  PROC DrawPart242()
    MoveL Offs(pOrigin,242.99,335.65,0.00),v40,z0,tPen\WObj:=wPaper;
    MoveL Offs(pOrigin,241.50,335.65,0.00),v40,fine,tPen\WObj:=wPaper;
    MoveL Offs(pOrigin,241.50,335.65,6.00),v60,z5,tPen\WObj:=wPaper;
    MoveL Offs(pOrigin,240.78,337.99,6.00),vTravel,z5,tPen\WObj:=wPaper;
    MoveL Offs(pOrigin,240.78,337.99,0.00),v60,z0,tPen\WObj:=wPaper;
    MoveL Offs(pOrigin,240.78,339.05,0.00),v40,z0,tPen\WObj:=wPaper;
    MoveL Offs(pOrigin,239.73,339.05,0.00),v40,z0,tPen\WObj:=wPaper;
    MoveL Offs(pOrigin,239.73,337.99,0.00),v40,fine,tPen\WObj:=wPaper;
    MoveL Offs(pOrigin,239.73,337.99,6.00),v60,z5,tPen\WObj:=wPaper;
    MoveL Offs(pOrigin,237.46,338.14,6.00),vTravel,z5,tPen\WObj:=wPaper;
    MoveL Offs(pOrigin,237.46,338.14,0.00),v60,z0,tPen\WObj:=wPaper;
    MoveL Offs(pOrigin,243.84,338.14,0.00),v40,fine,tPen\WObj:=wPaper;
    MoveL Offs(pOrigin,243.84,338.14,6.00),v60,z5,tPen\WObj:=wPaper;
    MoveL Offs(pOrigin,249.21,337.62,6.00),vTravel,z5,tPen\WObj:=wPaper;
    MoveL Offs(pOrigin,249.21,337.62,0.00),v60,z0,tPen\WObj:=wPaper;
    MoveL Offs(pOrigin,251.17,339.57,0.00),v40,fine,tPen\WObj:=wPaper;
    MoveL Offs(pOrigin,251.17,339.57,6.00),v60,z5,tPen\WObj:=wPaper;
    MoveL Offs(pOrigin,257.20,338.92,6.00),vTravel,z5,tPen\WObj:=wPaper;
    MoveL Offs(pOrigin,257.20,338.92,0.00),v60,z0,tPen\WObj:=wPaper;
    MoveL Offs(pOrigin,264.41,331.71,0.00),v40,fine,tPen\WObj:=wPaper;
    MoveL Offs(pOrigin,264.41,331.71,6.00),v60,z5,tPen\WObj:=wPaper;
    MoveL Offs(pOrigin,262.96,331.61,6.00),vTravel,z5,tPen\WObj:=wPaper;
    MoveL Offs(pOrigin,262.96,331.61,0.00),v60,z0,tPen\WObj:=wPaper;
    MoveL Offs(pOrigin,262.54,331.83,0.00),v40,z0,tPen\WObj:=wPaper;
    MoveL Offs(pOrigin,262.54,332.67,0.00),v40,fine,tPen\WObj:=wPaper;
    MoveL Offs(pOrigin,262.54,332.67,6.00),v60,z5,tPen\WObj:=wPaper;
    MoveL Offs(pOrigin,258.92,334.38,6.00),vTravel,z5,tPen\WObj:=wPaper;
    MoveL Offs(pOrigin,258.92,334.38,0.00),v60,z0,tPen\WObj:=wPaper;
    MoveL Offs(pOrigin,259.14,333.95,0.00),v40,z0,tPen\WObj:=wPaper;
    MoveL Offs(pOrigin,258.92,334.38,0.00),v40,z0,tPen\WObj:=wPaper;
    MoveL Offs(pOrigin,258.49,334.95,0.00),v40,z0,tPen\WObj:=wPaper;
    MoveL Offs(pOrigin,256.69,333.15,0.00),v40,fine,tPen\WObj:=wPaper;
    MoveL Offs(pOrigin,256.69,333.15,6.00),v60,z5,tPen\WObj:=wPaper;
    MoveL Offs(pOrigin,259.60,338.01,6.00),vTravel,z5,tPen\WObj:=wPaper;
    MoveL Offs(pOrigin,259.60,338.01,0.00),v60,z0,tPen\WObj:=wPaper;
    MoveL Offs(pOrigin,274.17,323.44,0.00),v40,fine,tPen\WObj:=wPaper;
    MoveL Offs(pOrigin,274.17,323.44,6.00),v60,z5,tPen\WObj:=wPaper;
    MoveL Offs(pOrigin,279.11,319.08,6.00),vTravel,z5,tPen\WObj:=wPaper;
    MoveL Offs(pOrigin,279.11,319.08,0.00),v60,z0,tPen\WObj:=wPaper;
    MoveL Offs(pOrigin,279.54,319.29,0.00),v40,z0,tPen\WObj:=wPaper;
    MoveL Offs(pOrigin,279.11,319.08,0.00),v40,fine,tPen\WObj:=wPaper;
    MoveL Offs(pOrigin,279.11,319.08,6.00),v60,z5,tPen\WObj:=wPaper;
    MoveL Offs(pOrigin,282.73,312.27,6.00),vTravel,z5,tPen\WObj:=wPaper;
    MoveL Offs(pOrigin,282.73,312.27,0.00),v60,z0,tPen\WObj:=wPaper;
    MoveL Offs(pOrigin,285.70,312.06,0.00),v40,z0,tPen\WObj:=wPaper;
    MoveL Offs(pOrigin,285.98,311.67,0.00),v40,z0,tPen\WObj:=wPaper;
    MoveL Offs(pOrigin,287.19,312.87,0.00),v40,z0,tPen\WObj:=wPaper;
    MoveL Offs(pOrigin,286.29,313.46,0.00),v40,z0,tPen\WObj:=wPaper;
    MoveL Offs(pOrigin,285.54,312.71,0.00),v40,fine,tPen\WObj:=wPaper;
    MoveL Offs(pOrigin,285.54,312.71,6.00),v60,z5,tPen\WObj:=wPaper;
    MoveL Offs(pOrigin,287.03,309.72,6.00),vTravel,z5,tPen\WObj:=wPaper;
    MoveL Offs(pOrigin,287.03,309.72,0.00),v60,z0,tPen\WObj:=wPaper;
    MoveL Offs(pOrigin,291.83,314.53,0.00),v40,fine,tPen\WObj:=wPaper;
    MoveL Offs(pOrigin,291.83,314.53,6.00),v60,z5,tPen\WObj:=wPaper;
    MoveL Offs(pOrigin,291.86,312.79,6.00),vTravel,z5,tPen\WObj:=wPaper;
    MoveL Offs(pOrigin,291.86,312.79,0.00),v60,z0,tPen\WObj:=wPaper;
    MoveL Offs(pOrigin,289.52,312.79,0.00),v40,z0,tPen\WObj:=wPaper;
    MoveL Offs(pOrigin,289.52,312.06,0.00),v40,z0,tPen\WObj:=wPaper;
    MoveL Offs(pOrigin,289.31,312.49,0.00),v40,z0,tPen\WObj:=wPaper;
    MoveL Offs(pOrigin,289.52,312.06,0.00),v40,z0,tPen\WObj:=wPaper;
    MoveL Offs(pOrigin,288.67,311.42,0.00),v40,z0,tPen\WObj:=wPaper;
    MoveL Offs(pOrigin,288.46,311.85,0.00),v40,z0,tPen\WObj:=wPaper;
    MoveL Offs(pOrigin,288.67,311.42,0.00),v40,fine,tPen\WObj:=wPaper;
    MoveL Offs(pOrigin,288.67,311.42,6.00),v60,z5,tPen\WObj:=wPaper;
    MoveL Offs(pOrigin,280.81,308.45,6.00),vTravel,z5,tPen\WObj:=wPaper;
    MoveL Offs(pOrigin,280.81,308.45,0.00),v60,z0,tPen\WObj:=wPaper;
    MoveL Offs(pOrigin,280.17,308.66,0.00),v40,z0,tPen\WObj:=wPaper;
    MoveL Offs(pOrigin,279.75,309.30,0.00),v40,z0,tPen\WObj:=wPaper;
    MoveL Offs(pOrigin,279.75,309.30,0.00),v40,z0,tPen\WObj:=wPaper;
    MoveL Offs(pOrigin,278.48,308.88,0.00),v40,z0,tPen\WObj:=wPaper;
    MoveL Offs(pOrigin,278.69,307.60,0.00),v40,z0,tPen\WObj:=wPaper;
    MoveL Offs(pOrigin,279.54,307.51,0.00),v40,z0,tPen\WObj:=wPaper;
    MoveL Offs(pOrigin,270.61,307.51,0.00),v40,fine,tPen\WObj:=wPaper;
    MoveL Offs(pOrigin,270.61,307.51,6.00),v60,z5,tPen\WObj:=wPaper;
    MoveL Offs(pOrigin,273.80,305.40,6.00),vTravel,z5,tPen\WObj:=wPaper;
    MoveL Offs(pOrigin,273.80,305.40,0.00),v60,z0,tPen\WObj:=wPaper;
    MoveL Offs(pOrigin,279.54,305.40,0.00),v40,z0,tPen\WObj:=wPaper;
    MoveL Offs(pOrigin,279.75,304.34,0.00),v40,z0,tPen\WObj:=wPaper;
    MoveL Offs(pOrigin,274.23,304.34,0.00),v40,fine,tPen\WObj:=wPaper;
    MoveL Offs(pOrigin,274.23,304.34,6.00),v60,z5,tPen\WObj:=wPaper;
    MoveL Offs(pOrigin,274.27,302.94,6.00),vTravel,z5,tPen\WObj:=wPaper;
    MoveL Offs(pOrigin,274.27,302.94,0.00),v60,z0,tPen\WObj:=wPaper;
    MoveL Offs(pOrigin,280.28,308.95,0.00),v40,fine,tPen\WObj:=wPaper;
    MoveL Offs(pOrigin,280.28,308.95,6.00),v60,z5,tPen\WObj:=wPaper;
    MoveL Offs(pOrigin,278.80,303.35,6.00),vTravel,z5,tPen\WObj:=wPaper;
    MoveL Offs(pOrigin,278.80,303.35,0.00),v60,z0,tPen\WObj:=wPaper;
    MoveL Offs(pOrigin,278.80,301.86,0.00),v40,fine,tPen\WObj:=wPaper;
    MoveL Offs(pOrigin,278.80,301.86,6.00),v60,z5,tPen\WObj:=wPaper;
    MoveL Offs(pOrigin,276.77,302.71,6.00),vTravel,z5,tPen\WObj:=wPaper;
    MoveL Offs(pOrigin,276.77,302.71,0.00),v60,z0,tPen\WObj:=wPaper;
    MoveL Offs(pOrigin,276.56,304.41,0.00),v40,fine,tPen\WObj:=wPaper;
    MoveL Offs(pOrigin,276.56,304.41,6.00),v60,z5,tPen\WObj:=wPaper;
    MoveL Offs(pOrigin,264.66,324.60,6.00),vTravel,z5,tPen\WObj:=wPaper;
    MoveL Offs(pOrigin,264.66,324.60,0.00),v60,z0,tPen\WObj:=wPaper;
    MoveL Offs(pOrigin,265.09,325.24,0.00),v40,z0,tPen\WObj:=wPaper;
    MoveL Offs(pOrigin,264.66,324.60,0.00),v40,fine,tPen\WObj:=wPaper;
    MoveL Offs(pOrigin,264.66,324.60,6.00),v60,z5,tPen\WObj:=wPaper;
    MoveL Offs(pOrigin,247.24,328.17,6.00),vTravel,z5,tPen\WObj:=wPaper;
    MoveL Offs(pOrigin,247.24,328.17,0.00),v60,z0,tPen\WObj:=wPaper;
    MoveL Offs(pOrigin,232.66,313.60,0.00),v40,fine,tPen\WObj:=wPaper;
    MoveL Offs(pOrigin,232.66,313.60,6.00),v60,z5,tPen\WObj:=wPaper;
    MoveL Offs(pOrigin,231.09,314.90,6.00),vTravel,z5,tPen\WObj:=wPaper;
    MoveL Offs(pOrigin,231.09,314.90,0.00),v60,z0,tPen\WObj:=wPaper;
    MoveL Offs(pOrigin,216.64,314.90,0.00),v40,z0,tPen\WObj:=wPaper;
    MoveL Offs(pOrigin,216.64,315.67,0.00),v40,z0,tPen\WObj:=wPaper;
    MoveL Offs(pOrigin,216.00,316.10,0.00),v40,z0,tPen\WObj:=wPaper;
    MoveL Offs(pOrigin,215.72,317.38,0.00),v40,z0,tPen\WObj:=wPaper;
    MoveL Offs(pOrigin,215.15,317.80,0.00),v40,fine,tPen\WObj:=wPaper;
    MoveL Offs(pOrigin,215.15,317.80,6.00),v60,z5,tPen\WObj:=wPaper;
    MoveL Offs(pOrigin,213.95,317.29,6.00),vTravel,z5,tPen\WObj:=wPaper;
    MoveL Offs(pOrigin,213.95,317.29,0.00),v60,z0,tPen\WObj:=wPaper;
    MoveL Offs(pOrigin,210.34,313.68,0.00),v40,z0,tPen\WObj:=wPaper;
    MoveL Offs(pOrigin,210.05,313.76,0.00),v40,z0,tPen\WObj:=wPaper;
    MoveL Offs(pOrigin,209.62,314.19,0.00),v40,z0,tPen\WObj:=wPaper;
    MoveL Offs(pOrigin,210.05,313.76,0.00),v40,fine,tPen\WObj:=wPaper;
    MoveL Offs(pOrigin,210.05,313.76,6.00),v60,z5,tPen\WObj:=wPaper;
    MoveL Offs(pOrigin,210.90,312.91,6.00),vTravel,z5,tPen\WObj:=wPaper;
    MoveL Offs(pOrigin,210.90,312.91,0.00),v60,z0,tPen\WObj:=wPaper;
    MoveL Offs(pOrigin,210.26,313.55,0.00),v40,z0,tPen\WObj:=wPaper;
    MoveL Offs(pOrigin,210.90,312.91,0.00),v40,z0,tPen\WObj:=wPaper;
  ENDPROC

  PROC DrawPart243()
    MoveL Offs(pOrigin,210.94,312.78,0.00),v40,z0,tPen\WObj:=wPaper;
    MoveL Offs(pOrigin,214.69,316.54,0.00),v40,fine,tPen\WObj:=wPaper;
    MoveL Offs(pOrigin,214.69,316.54,6.00),v60,z5,tPen\WObj:=wPaper;
    MoveL Offs(pOrigin,213.45,317.02,6.00),vTravel,z5,tPen\WObj:=wPaper;
    MoveL Offs(pOrigin,213.45,317.02,0.00),v60,z0,tPen\WObj:=wPaper;
    MoveL Offs(pOrigin,212.39,317.02,0.00),v40,z0,tPen\WObj:=wPaper;
    MoveL Offs(pOrigin,211.85,316.68,0.00),v40,z0,tPen\WObj:=wPaper;
    MoveL Offs(pOrigin,213.50,318.33,0.00),v40,z0,tPen\WObj:=wPaper;
    MoveL Offs(pOrigin,213.24,318.07,0.00),v40,z0,tPen\WObj:=wPaper;
    MoveL Offs(pOrigin,211.96,318.07,0.00),v40,z0,tPen\WObj:=wPaper;
    MoveL Offs(pOrigin,211.55,317.88,0.00),v40,z0,tPen\WObj:=wPaper;
    MoveL Offs(pOrigin,213.21,319.53,0.00),v40,z0,tPen\WObj:=wPaper;
    MoveL Offs(pOrigin,212.81,319.13,0.00),v40,z0,tPen\WObj:=wPaper;
    MoveL Offs(pOrigin,211.32,319.13,0.00),v40,z0,tPen\WObj:=wPaper;
    MoveL Offs(pOrigin,211.32,319.08,0.00),v40,z0,tPen\WObj:=wPaper;
    MoveL Offs(pOrigin,211.54,318.65,0.00),v40,z0,tPen\WObj:=wPaper;
    MoveL Offs(pOrigin,211.32,319.08,0.00),v40,z0,tPen\WObj:=wPaper;
    MoveL Offs(pOrigin,210.96,318.77,0.00),v40,z0,tPen\WObj:=wPaper;
    MoveL Offs(pOrigin,212.76,320.58,0.00),v40,fine,tPen\WObj:=wPaper;
    MoveL Offs(pOrigin,212.76,320.58,6.00),v60,z5,tPen\WObj:=wPaper;
    MoveL Offs(pOrigin,210.21,323.19,6.00),vTravel,z5,tPen\WObj:=wPaper;
    MoveL Offs(pOrigin,210.21,323.19,0.00),v60,z0,tPen\WObj:=wPaper;
    MoveL Offs(pOrigin,204.35,329.05,0.00),v40,fine,tPen\WObj:=wPaper;
    MoveL Offs(pOrigin,204.35,329.05,6.00),v60,z5,tPen\WObj:=wPaper;
    MoveL Offs(pOrigin,208.05,327.15,6.00),vTravel,z5,tPen\WObj:=wPaper;
    MoveL Offs(pOrigin,208.05,327.15,0.00),v60,z0,tPen\WObj:=wPaper;
    MoveL Offs(pOrigin,208.05,325.88,0.00),v40,fine,tPen\WObj:=wPaper;
    MoveL Offs(pOrigin,208.05,325.88,6.00),v60,z5,tPen\WObj:=wPaper;
    MoveL Offs(pOrigin,209.10,326.51,6.00),vTravel,z5,tPen\WObj:=wPaper;
    MoveL Offs(pOrigin,209.10,326.51,0.00),v60,z0,tPen\WObj:=wPaper;
    MoveL Offs(pOrigin,209.10,327.58,0.00),v40,fine,tPen\WObj:=wPaper;
    MoveL Offs(pOrigin,209.10,327.58,6.00),v60,z5,tPen\WObj:=wPaper;
    MoveL Offs(pOrigin,210.26,329.06,6.00),vTravel,z5,tPen\WObj:=wPaper;
    MoveL Offs(pOrigin,210.26,329.06,0.00),v60,z0,tPen\WObj:=wPaper;
    MoveL Offs(pOrigin,210.69,329.49,0.00),v40,z0,tPen\WObj:=wPaper;
    MoveL Offs(pOrigin,210.26,329.06,0.00),v40,fine,tPen\WObj:=wPaper;
    MoveL Offs(pOrigin,210.26,329.06,6.00),v60,z5,tPen\WObj:=wPaper;
    MoveL Offs(pOrigin,209.41,325.66,6.00),vTravel,z5,tPen\WObj:=wPaper;
    MoveL Offs(pOrigin,209.41,325.66,0.00),v60,z0,tPen\WObj:=wPaper;
    MoveL Offs(pOrigin,209.84,326.09,0.00),v40,z0,tPen\WObj:=wPaper;
    MoveL Offs(pOrigin,209.41,325.66,0.00),v40,z0,tPen\WObj:=wPaper;
    MoveL Offs(pOrigin,209.93,325.21,0.00),v40,z0,tPen\WObj:=wPaper;
    MoveL Offs(pOrigin,209.03,324.31,0.00),v40,fine,tPen\WObj:=wPaper;
    MoveL Offs(pOrigin,209.03,324.31,6.00),v60,z5,tPen\WObj:=wPaper;
    MoveL Offs(pOrigin,214.88,327.18,6.00),vTravel,z5,tPen\WObj:=wPaper;
    MoveL Offs(pOrigin,214.88,327.18,0.00),v60,z0,tPen\WObj:=wPaper;
    MoveL Offs(pOrigin,217.13,329.43,0.00),v40,fine,tPen\WObj:=wPaper;
    MoveL Offs(pOrigin,217.13,329.43,6.00),v60,z5,tPen\WObj:=wPaper;
    MoveL Offs(pOrigin,219.38,328.69,6.00),vTravel,z5,tPen\WObj:=wPaper;
    MoveL Offs(pOrigin,219.38,328.69,0.00),v60,z0,tPen\WObj:=wPaper;
    MoveL Offs(pOrigin,217.72,327.03,0.00),v40,fine,tPen\WObj:=wPaper;
    MoveL Offs(pOrigin,217.72,327.03,6.00),v60,z5,tPen\WObj:=wPaper;
    MoveL Offs(pOrigin,220.68,328.42,6.00),vTravel,z5,tPen\WObj:=wPaper;
    MoveL Offs(pOrigin,220.68,328.42,0.00),v60,z0,tPen\WObj:=wPaper;
    MoveL Offs(pOrigin,221.10,328.21,0.00),v40,z0,tPen\WObj:=wPaper;
    MoveL Offs(pOrigin,220.68,328.42,0.00),v40,fine,tPen\WObj:=wPaper;
    MoveL Offs(pOrigin,220.68,328.42,6.00),v60,z5,tPen\WObj:=wPaper;
    MoveL Offs(pOrigin,223.12,329.45,6.00),vTravel,z5,tPen\WObj:=wPaper;
    MoveL Offs(pOrigin,223.12,329.45,0.00),v60,z0,tPen\WObj:=wPaper;
    MoveL Offs(pOrigin,224.17,330.50,0.00),v40,z0,tPen\WObj:=wPaper;
    MoveL Offs(pOrigin,224.77,329.60,0.00),v40,z0,tPen\WObj:=wPaper;
    MoveL Offs(pOrigin,223.87,328.70,0.00),v40,z0,tPen\WObj:=wPaper;
    MoveL Offs(pOrigin,224.71,329.06,0.00),v40,z0,tPen\WObj:=wPaper;
    MoveL Offs(pOrigin,223.44,329.06,0.00),v40,z0,tPen\WObj:=wPaper;
    MoveL Offs(pOrigin,219.61,330.55,0.00),v40,z0,tPen\WObj:=wPaper;
    MoveL Offs(pOrigin,216.21,330.76,0.00),v40,z0,tPen\WObj:=wPaper;
    MoveL Offs(pOrigin,215.86,330.98,0.00),v40,z0,tPen\WObj:=wPaper;
    MoveL Offs(pOrigin,215.79,331.61,0.00),v40,fine,tPen\WObj:=wPaper;
    MoveL Offs(pOrigin,215.79,331.61,6.00),v60,z5,tPen\WObj:=wPaper;
    MoveL Offs(pOrigin,215.58,332.86,6.00),vTravel,z5,tPen\WObj:=wPaper;
    MoveL Offs(pOrigin,215.58,332.86,0.00),v60,z0,tPen\WObj:=wPaper;
    MoveL Offs(pOrigin,214.51,332.86,0.00),v40,fine,tPen\WObj:=wPaper;
    MoveL Offs(pOrigin,214.51,332.86,6.00),v60,z5,tPen\WObj:=wPaper;
    MoveL Offs(pOrigin,209.20,333.52,6.00),vTravel,z5,tPen\WObj:=wPaper;
    MoveL Offs(pOrigin,209.20,333.52,0.00),v60,z0,tPen\WObj:=wPaper;
    MoveL Offs(pOrigin,209.62,333.74,0.00),v40,z0,tPen\WObj:=wPaper;
    MoveL Offs(pOrigin,209.20,333.52,0.00),v40,fine,tPen\WObj:=wPaper;
    MoveL Offs(pOrigin,209.20,333.52,6.00),v60,z5,tPen\WObj:=wPaper;
    MoveL Offs(pOrigin,218.86,336.94,6.00),vTravel,z5,tPen\WObj:=wPaper;
    MoveL Offs(pOrigin,218.86,336.94,0.00),v60,z0,tPen\WObj:=wPaper;
    MoveL Offs(pOrigin,226.67,329.13,0.00),v40,z0,tPen\WObj:=wPaper;
    MoveL Offs(pOrigin,227.05,328.00,0.00),v40,z0,tPen\WObj:=wPaper;
    MoveL Offs(pOrigin,227.26,327.58,0.00),v40,z0,tPen\WObj:=wPaper;
    MoveL Offs(pOrigin,227.05,328.00,0.00),v40,fine,tPen\WObj:=wPaper;
    MoveL Offs(pOrigin,227.05,328.00,6.00),v60,z5,tPen\WObj:=wPaper;
    MoveL Offs(pOrigin,228.02,329.27,6.00),vTravel,z5,tPen\WObj:=wPaper;
    MoveL Offs(pOrigin,228.02,329.27,0.00),v60,z0,tPen\WObj:=wPaper;
    MoveL Offs(pOrigin,220.20,337.09,0.00),v40,fine,tPen\WObj:=wPaper;
    MoveL Offs(pOrigin,220.20,337.09,6.00),v60,z5,tPen\WObj:=wPaper;
    MoveL Offs(pOrigin,226.41,336.02,6.00),vTravel,z5,tPen\WObj:=wPaper;
    MoveL Offs(pOrigin,226.41,336.02,0.00),v60,z0,tPen\WObj:=wPaper;
    MoveL Offs(pOrigin,232.79,336.02,0.00),v40,fine,tPen\WObj:=wPaper;
    MoveL Offs(pOrigin,232.79,336.02,6.00),v60,z5,tPen\WObj:=wPaper;
    MoveL Offs(pOrigin,233.10,333.15,6.00),vTravel,z5,tPen\WObj:=wPaper;
    MoveL Offs(pOrigin,233.10,333.15,0.00),v60,z0,tPen\WObj:=wPaper;
    MoveL Offs(pOrigin,226.64,339.61,0.00),v40,fine,tPen\WObj:=wPaper;
    MoveL Offs(pOrigin,226.64,339.61,6.00),v60,z5,tPen\WObj:=wPaper;
    MoveL Offs(pOrigin,226.00,333.31,6.00),vTravel,z5,tPen\WObj:=wPaper;
    MoveL Offs(pOrigin,226.00,333.31,0.00),v60,z0,tPen\WObj:=wPaper;
    MoveL Offs(pOrigin,226.00,332.04,0.00),v40,z0,tPen\WObj:=wPaper;
    MoveL Offs(pOrigin,226.27,331.11,0.00),v40,z0,tPen\WObj:=wPaper;
    MoveL Offs(pOrigin,228.38,333.21,0.00),v40,fine,tPen\WObj:=wPaper;
    MoveL Offs(pOrigin,228.38,333.21,6.00),v60,z5,tPen\WObj:=wPaper;
    MoveL Offs(pOrigin,224.73,326.59,6.00),vTravel,z5,tPen\WObj:=wPaper;
    MoveL Offs(pOrigin,224.73,326.59,0.00),v60,z0,tPen\WObj:=wPaper;
    MoveL Offs(pOrigin,240.51,310.81,0.00),v40,fine,tPen\WObj:=wPaper;
    MoveL Offs(pOrigin,240.51,310.81,6.00),v60,z5,tPen\WObj:=wPaper;
    MoveL Offs(pOrigin,238.20,313.17,6.00),vTravel,z5,tPen\WObj:=wPaper;
    MoveL Offs(pOrigin,238.20,313.17,0.00),v60,z0,tPen\WObj:=wPaper;
    MoveL Offs(pOrigin,239.25,314.22,0.00),v40,fine,tPen\WObj:=wPaper;
    MoveL Offs(pOrigin,239.25,314.22,6.00),v60,z5,tPen\WObj:=wPaper;
    MoveL Offs(pOrigin,244.19,313.18,6.00),vTravel,z5,tPen\WObj:=wPaper;
    MoveL Offs(pOrigin,244.19,313.18,0.00),v60,z0,tPen\WObj:=wPaper;
    MoveL Offs(pOrigin,245.25,314.24,0.00),v40,fine,tPen\WObj:=wPaper;
    MoveL Offs(pOrigin,245.25,314.24,6.00),v60,z5,tPen\WObj:=wPaper;
    MoveL Offs(pOrigin,234.45,320.77,6.00),vTravel,z5,tPen\WObj:=wPaper;
    MoveL Offs(pOrigin,234.45,320.77,0.00),v60,z0,tPen\WObj:=wPaper;
    MoveL Offs(pOrigin,234.45,322.90,0.00),v40,fine,tPen\WObj:=wPaper;
    MoveL Offs(pOrigin,234.45,322.90,6.00),v60,z5,tPen\WObj:=wPaper;
    MoveL Offs(pOrigin,233.00,318.07,6.00),vTravel,z5,tPen\WObj:=wPaper;
  ENDPROC

  PROC DrawPart244()
    MoveL Offs(pOrigin,233.00,318.07,0.00),v60,z0,tPen\WObj:=wPaper;
    MoveL Offs(pOrigin,217.91,318.07,0.00),v40,z0,tPen\WObj:=wPaper;
    MoveL Offs(pOrigin,217.70,317.02,0.00),v40,z0,tPen\WObj:=wPaper;
    MoveL Offs(pOrigin,231.94,317.02,0.00),v40,z0,tPen\WObj:=wPaper;
    MoveL Offs(pOrigin,231.30,317.80,0.00),v40,z0,tPen\WObj:=wPaper;
    MoveL Offs(pOrigin,231.09,316.52,0.00),v40,z0,tPen\WObj:=wPaper;
    MoveL Offs(pOrigin,230.45,316.10,0.00),v40,fine,tPen\WObj:=wPaper;
    MoveL Offs(pOrigin,230.45,316.10,6.00),v60,z5,tPen\WObj:=wPaper;
    MoveL Offs(pOrigin,226.00,314.82,6.00),vTravel,z5,tPen\WObj:=wPaper;
    MoveL Offs(pOrigin,226.00,314.82,0.00),v60,z0,tPen\WObj:=wPaper;
    MoveL Offs(pOrigin,226.00,317.80,0.00),v40,fine,tPen\WObj:=wPaper;
    MoveL Offs(pOrigin,226.00,317.80,6.00),v60,z5,tPen\WObj:=wPaper;
    MoveL Offs(pOrigin,221.31,313.34,6.00),vTravel,z5,tPen\WObj:=wPaper;
    MoveL Offs(pOrigin,221.31,313.34,0.00),v60,z0,tPen\WObj:=wPaper;
    MoveL Offs(pOrigin,221.74,312.06,0.00),v40,z0,tPen\WObj:=wPaper;
    MoveL Offs(pOrigin,221.52,311.71,0.00),v40,z0,tPen\WObj:=wPaper;
    MoveL Offs(pOrigin,220.46,312.06,0.00),v40,z0,tPen\WObj:=wPaper;
    MoveL Offs(pOrigin,219.61,313.34,0.00),v40,fine,tPen\WObj:=wPaper;
    MoveL Offs(pOrigin,219.61,313.34,6.00),v60,z5,tPen\WObj:=wPaper;
    MoveL Offs(pOrigin,216.64,313.98,6.00),vTravel,z5,tPen\WObj:=wPaper;
    MoveL Offs(pOrigin,216.64,313.98,0.00),v60,z0,tPen\WObj:=wPaper;
    MoveL Offs(pOrigin,215.57,313.55,0.00),v40,z0,tPen\WObj:=wPaper;
    MoveL Offs(pOrigin,215.57,313.55,0.00),v40,z0,tPen\WObj:=wPaper;
    MoveL Offs(pOrigin,216.00,312.06,0.00),v40,z0,tPen\WObj:=wPaper;
    MoveL Offs(pOrigin,216.64,311.64,0.00),v40,z0,tPen\WObj:=wPaper;
    MoveL Offs(pOrigin,216.21,312.06,0.00),v40,z0,tPen\WObj:=wPaper;
    MoveL Offs(pOrigin,216.64,311.64,0.00),v40,z0,tPen\WObj:=wPaper;
    MoveL Offs(pOrigin,216.21,312.06,0.00),v40,z0,tPen\WObj:=wPaper;
    MoveL Offs(pOrigin,215.44,311.64,0.00),v40,z0,tPen\WObj:=wPaper;
    MoveL Offs(pOrigin,215.44,309.30,0.00),v40,z0,tPen\WObj:=wPaper;
    MoveL Offs(pOrigin,216.49,308.88,0.00),v40,z0,tPen\WObj:=wPaper;
    MoveL Offs(pOrigin,216.49,311.00,0.00),v40,fine,tPen\WObj:=wPaper;
    MoveL Offs(pOrigin,216.49,311.00,6.00),v60,z5,tPen\WObj:=wPaper;
    MoveL Offs(pOrigin,214.38,310.79,6.00),vTravel,z5,tPen\WObj:=wPaper;
    MoveL Offs(pOrigin,214.38,310.79,0.00),v60,z0,tPen\WObj:=wPaper;
    MoveL Offs(pOrigin,214.38,313.12,0.00),v40,fine,tPen\WObj:=wPaper;
    MoveL Offs(pOrigin,214.38,313.12,6.00),v60,z5,tPen\WObj:=wPaper;
    MoveL Offs(pOrigin,213.33,309.30,6.00),vTravel,z5,tPen\WObj:=wPaper;
    MoveL Offs(pOrigin,213.33,309.30,0.00),v60,z0,tPen\WObj:=wPaper;
    MoveL Offs(pOrigin,213.33,306.96,0.00),v40,z0,tPen\WObj:=wPaper;
    MoveL Offs(pOrigin,212.27,306.75,0.00),v40,z0,tPen\WObj:=wPaper;
    MoveL Offs(pOrigin,212.27,308.66,0.00),v40,z0,tPen\WObj:=wPaper;
    MoveL Offs(pOrigin,211.21,308.45,0.00),v40,z0,tPen\WObj:=wPaper;
    MoveL Offs(pOrigin,211.21,306.32,0.00),v40,z0,tPen\WObj:=wPaper;
    MoveL Offs(pOrigin,210.69,306.96,0.00),v40,z0,tPen\WObj:=wPaper;
    MoveL Offs(pOrigin,211.96,306.75,0.00),v40,z0,tPen\WObj:=wPaper;
    MoveL Offs(pOrigin,212.81,305.97,0.00),v40,z0,tPen\WObj:=wPaper;
    MoveL Offs(pOrigin,213.88,305.69,0.00),v40,fine,tPen\WObj:=wPaper;
    MoveL Offs(pOrigin,213.88,305.69,6.00),v60,z5,tPen\WObj:=wPaper;
    MoveL Offs(pOrigin,211.96,303.35,6.00),vTravel,z5,tPen\WObj:=wPaper;
    MoveL Offs(pOrigin,211.96,303.35,0.00),v60,z0,tPen\WObj:=wPaper;
    MoveL Offs(pOrigin,211.47,301.86,0.00),v40,z0,tPen\WObj:=wPaper;
    MoveL Offs(pOrigin,209.84,301.01,0.00),v40,z0,tPen\WObj:=wPaper;
    MoveL Offs(pOrigin,209.84,301.01,0.00),v40,z0,tPen\WObj:=wPaper;
    MoveL Offs(pOrigin,207.93,300.66,0.00),v40,z0,tPen\WObj:=wPaper;
    MoveL Offs(pOrigin,207.29,300.02,0.00),v40,z0,tPen\WObj:=wPaper;
    MoveL Offs(pOrigin,205.80,300.23,0.00),v40,z0,tPen\WObj:=wPaper;
    MoveL Offs(pOrigin,202.82,298.53,0.00),v40,z0,tPen\WObj:=wPaper;
    MoveL Offs(pOrigin,202.40,298.89,0.00),v40,z0,tPen\WObj:=wPaper;
    MoveL Offs(pOrigin,202.40,299.95,0.00),v40,z0,tPen\WObj:=wPaper;
    MoveL Offs(pOrigin,203.04,300.12,0.00),v40,z0,tPen\WObj:=wPaper;
    MoveL Offs(pOrigin,208.78,300.12,0.00),v40,fine,tPen\WObj:=wPaper;
    MoveL Offs(pOrigin,208.78,300.12,6.00),v60,z5,tPen\WObj:=wPaper;
    MoveL Offs(pOrigin,209.84,301.01,6.00),vTravel,z5,tPen\WObj:=wPaper;
    MoveL Offs(pOrigin,209.84,301.01,0.00),v60,z0,tPen\WObj:=wPaper;
    MoveL Offs(pOrigin,209.34,298.89,0.00),v40,z0,tPen\WObj:=wPaper;
    MoveL Offs(pOrigin,207.50,296.76,0.00),v40,fine,tPen\WObj:=wPaper;
    MoveL Offs(pOrigin,207.50,296.76,6.00),v60,z5,tPen\WObj:=wPaper;
    MoveL Offs(pOrigin,205.59,302.92,6.00),vTravel,z5,tPen\WObj:=wPaper;
    MoveL Offs(pOrigin,205.59,302.92,0.00),v60,z0,tPen\WObj:=wPaper;
    MoveL Offs(pOrigin,206.65,303.14,0.00),v40,z0,tPen\WObj:=wPaper;
    MoveL Offs(pOrigin,206.86,303.77,0.00),v40,fine,tPen\WObj:=wPaper;
    MoveL Offs(pOrigin,206.86,303.77,6.00),v60,z5,tPen\WObj:=wPaper;
    MoveL Offs(pOrigin,202.24,308.56,6.00),vTravel,z5,tPen\WObj:=wPaper;
    MoveL Offs(pOrigin,202.24,308.56,0.00),v60,z0,tPen\WObj:=wPaper;
    MoveL Offs(pOrigin,200.13,306.46,0.00),v40,z0,tPen\WObj:=wPaper;
    MoveL Offs(pOrigin,199.21,306.46,0.00),v40,z0,tPen\WObj:=wPaper;
    MoveL Offs(pOrigin,197.51,306.46,0.00),v40,fine,tPen\WObj:=wPaper;
    MoveL Offs(pOrigin,197.51,306.46,6.00),v60,z5,tPen\WObj:=wPaper;
    MoveL Offs(pOrigin,199.64,300.59,6.00),vTravel,z5,tPen\WObj:=wPaper;
    MoveL Offs(pOrigin,199.64,300.59,0.00),v60,z0,tPen\WObj:=wPaper;
    MoveL Offs(pOrigin,200.06,300.80,0.00),v40,z0,tPen\WObj:=wPaper;
    MoveL Offs(pOrigin,199.64,300.59,0.00),v40,fine,tPen\WObj:=wPaper;
    MoveL Offs(pOrigin,199.64,300.59,6.00),v60,z5,tPen\WObj:=wPaper;
    MoveL Offs(pOrigin,207.95,315.77,6.00),vTravel,z5,tPen\WObj:=wPaper;
    MoveL Offs(pOrigin,207.95,315.77,0.00),v60,z0,tPen\WObj:=wPaper;
    MoveL Offs(pOrigin,209.00,316.82,0.00),v40,z0,tPen\WObj:=wPaper;
    MoveL Offs(pOrigin,209.20,316.95,0.00),v40,z0,tPen\WObj:=wPaper;
    MoveL Offs(pOrigin,208.92,317.52,0.00),v40,z0,tPen\WObj:=wPaper;
    MoveL Offs(pOrigin,207.50,318.01,0.00),v40,z0,tPen\WObj:=wPaper;
    MoveL Offs(pOrigin,205.59,318.23,0.00),v40,z0,tPen\WObj:=wPaper;
    MoveL Offs(pOrigin,202.19,317.80,0.00),v40,z0,tPen\WObj:=wPaper;
    MoveL Offs(pOrigin,201.76,318.01,0.00),v40,fine,tPen\WObj:=wPaper;
    MoveL Offs(pOrigin,201.76,318.01,6.00),v60,z5,tPen\WObj:=wPaper;
    MoveL Offs(pOrigin,219.66,319.29,6.00),vTravel,z5,tPen\WObj:=wPaper;
    MoveL Offs(pOrigin,219.66,319.29,0.00),v60,z0,tPen\WObj:=wPaper;
    MoveL Offs(pOrigin,219.66,309.94,0.00),v40,fine,tPen\WObj:=wPaper;
    MoveL Offs(pOrigin,219.66,309.94,6.00),v60,z5,tPen\WObj:=wPaper;
    MoveL Offs(pOrigin,222.65,271.92,6.00),vTravel,z5,tPen\WObj:=wPaper;
    MoveL Offs(pOrigin,222.65,271.92,0.00),v60,z0,tPen\WObj:=wPaper;
    MoveL Offs(pOrigin,238.28,256.29,0.00),v40,fine,tPen\WObj:=wPaper;
    MoveL Offs(pOrigin,238.28,256.29,6.00),v60,z5,tPen\WObj:=wPaper;
    MoveL Offs(pOrigin,237.09,254.50,6.00),vTravel,z5,tPen\WObj:=wPaper;
    MoveL Offs(pOrigin,237.09,254.50,0.00),v60,z0,tPen\WObj:=wPaper;
    MoveL Offs(pOrigin,234.68,256.90,0.00),v40,z0,tPen\WObj:=wPaper;
    MoveL Offs(pOrigin,233.93,257.65,0.00),v40,z0,tPen\WObj:=wPaper;
    MoveL Offs(pOrigin,220.26,271.32,0.00),v40,z0,tPen\WObj:=wPaper;
    MoveL Offs(pOrigin,219.95,271.02,0.00),v40,z0,tPen\WObj:=wPaper;
    MoveL Offs(pOrigin,212.74,263.80,0.00),v40,z0,tPen\WObj:=wPaper;
    MoveL Offs(pOrigin,212.19,264.46,0.00),v40,z0,tPen\WObj:=wPaper;
    MoveL Offs(pOrigin,213.99,262.66,0.00),v40,z0,tPen\WObj:=wPaper;
    MoveL Offs(pOrigin,213.39,261.76,0.00),v40,z0,tPen\WObj:=wPaper;
    MoveL Offs(pOrigin,212.04,263.11,0.00),v40,fine,tPen\WObj:=wPaper;
    MoveL Offs(pOrigin,212.04,263.11,6.00),v60,z5,tPen\WObj:=wPaper;
    MoveL Offs(pOrigin,214.00,259.66,6.00),vTravel,z5,tPen\WObj:=wPaper;
    MoveL Offs(pOrigin,214.00,259.66,0.00),v60,z0,tPen\WObj:=wPaper;
    MoveL Offs(pOrigin,215.95,257.71,0.00),v40,fine,tPen\WObj:=wPaper;
    MoveL Offs(pOrigin,215.95,257.71,6.00),v60,z5,tPen\WObj:=wPaper;
    MoveL Offs(pOrigin,215.36,259.15,6.00),vTravel,z5,tPen\WObj:=wPaper;
    MoveL Offs(pOrigin,215.36,259.15,0.00),v60,z0,tPen\WObj:=wPaper;
  ENDPROC

  PROC DrawPart245()
    MoveL Offs(pOrigin,216.21,259.58,0.00),v40,z0,tPen\WObj:=wPaper;
    MoveL Offs(pOrigin,216.85,259.99,0.00),v40,z0,tPen\WObj:=wPaper;
    MoveL Offs(pOrigin,218.34,259.99,0.00),v40,z0,tPen\WObj:=wPaper;
    MoveL Offs(pOrigin,217.91,259.58,0.00),v40,z0,tPen\WObj:=wPaper;
    MoveL Offs(pOrigin,218.34,260.00,0.00),v40,z0,tPen\WObj:=wPaper;
    MoveL Offs(pOrigin,217.91,259.58,0.00),v40,fine,tPen\WObj:=wPaper;
    MoveL Offs(pOrigin,217.91,259.58,6.00),v60,z5,tPen\WObj:=wPaper;
    MoveL Offs(pOrigin,219.19,257.45,6.00),vTravel,z5,tPen\WObj:=wPaper;
    MoveL Offs(pOrigin,219.19,257.45,0.00),v60,z0,tPen\WObj:=wPaper;
    MoveL Offs(pOrigin,221.52,257.24,0.00),v40,fine,tPen\WObj:=wPaper;
    MoveL Offs(pOrigin,221.52,257.24,6.00),v60,z5,tPen\WObj:=wPaper;
    MoveL Offs(pOrigin,222.59,256.39,6.00),vTravel,z5,tPen\WObj:=wPaper;
    MoveL Offs(pOrigin,222.59,256.39,0.00),v60,z0,tPen\WObj:=wPaper;
    MoveL Offs(pOrigin,226.41,257.02,0.00),v40,z0,tPen\WObj:=wPaper;
    MoveL Offs(pOrigin,229.18,258.02,0.00),v40,z0,tPen\WObj:=wPaper;
    MoveL Offs(pOrigin,231.51,259.29,0.00),v40,z0,tPen\WObj:=wPaper;
    MoveL Offs(pOrigin,233.00,259.58,0.00),v40,z0,tPen\WObj:=wPaper;
    MoveL Offs(pOrigin,233.09,258.77,0.00),v40,z0,tPen\WObj:=wPaper;
    MoveL Offs(pOrigin,238.20,263.88,0.00),v40,z0,tPen\WObj:=wPaper;
    MoveL Offs(pOrigin,237.25,263.83,0.00),v40,z0,tPen\WObj:=wPaper;
    MoveL Offs(pOrigin,238.24,262.98,0.00),v40,z0,tPen\WObj:=wPaper;
    MoveL Offs(pOrigin,238.31,262.12,0.00),v40,z0,tPen\WObj:=wPaper;
    MoveL Offs(pOrigin,237.04,260.85,0.00),v40,z0,tPen\WObj:=wPaper;
    MoveL Offs(pOrigin,237.04,260.85,0.00),v40,z0,tPen\WObj:=wPaper;
    MoveL Offs(pOrigin,236.82,259.58,0.00),v40,z0,tPen\WObj:=wPaper;
    MoveL Offs(pOrigin,236.82,259.58,0.00),v40,z0,tPen\WObj:=wPaper;
    MoveL Offs(pOrigin,236.75,258.51,0.00),v40,z0,tPen\WObj:=wPaper;
    MoveL Offs(pOrigin,235.98,258.09,0.00),v40,z0,tPen\WObj:=wPaper;
    MoveL Offs(pOrigin,234.49,259.58,0.00),v40,z0,tPen\WObj:=wPaper;
    MoveL Offs(pOrigin,234.49,259.58,0.00),v40,z0,tPen\WObj:=wPaper;
    MoveL Offs(pOrigin,235.12,260.21,0.00),v40,z0,tPen\WObj:=wPaper;
    MoveL Offs(pOrigin,235.12,260.21,0.00),v40,z0,tPen\WObj:=wPaper;
    MoveL Offs(pOrigin,235.12,260.00,0.00),v40,z0,tPen\WObj:=wPaper;
    MoveL Offs(pOrigin,236.19,260.21,0.00),v40,z0,tPen\WObj:=wPaper;
    MoveL Offs(pOrigin,236.82,259.58,0.00),v40,z0,tPen\WObj:=wPaper;
    MoveL Offs(pOrigin,236.19,259.99,0.00),v40,z0,tPen\WObj:=wPaper;
    MoveL Offs(pOrigin,237.46,259.99,0.00),v40,z0,tPen\WObj:=wPaper;
    MoveL Offs(pOrigin,237.04,260.85,0.00),v40,z0,tPen\WObj:=wPaper;
    MoveL Offs(pOrigin,236.19,262.34,0.00),v40,z0,tPen\WObj:=wPaper;
    MoveL Offs(pOrigin,236.40,262.10,0.00),v40,z0,tPen\WObj:=wPaper;
    MoveL Offs(pOrigin,237.68,262.10,0.00),v40,z0,tPen\WObj:=wPaper;
    MoveL Offs(pOrigin,237.46,263.16,0.00),v40,z0,tPen\WObj:=wPaper;
    MoveL Offs(pOrigin,235.12,263.16,0.00),v40,z0,tPen\WObj:=wPaper;
    MoveL Offs(pOrigin,235.34,262.34,0.00),v40,z0,tPen\WObj:=wPaper;
    MoveL Offs(pOrigin,236.19,262.55,0.00),v40,z0,tPen\WObj:=wPaper;
    MoveL Offs(pOrigin,236.82,263.83,0.00),v40,fine,tPen\WObj:=wPaper;
    MoveL Offs(pOrigin,236.82,263.83,6.00),v60,z5,tPen\WObj:=wPaper;
    MoveL Offs(pOrigin,235.34,262.34,6.00),vTravel,z5,tPen\WObj:=wPaper;
    MoveL Offs(pOrigin,235.34,262.34,0.00),v60,z0,tPen\WObj:=wPaper;
    MoveL Offs(pOrigin,234.91,261.27,0.00),v40,z0,tPen\WObj:=wPaper;
    MoveL Offs(pOrigin,235.12,260.21,0.00),v40,z0,tPen\WObj:=wPaper;
    MoveL Offs(pOrigin,234.49,259.58,0.00),v40,z0,tPen\WObj:=wPaper;
    MoveL Offs(pOrigin,233.21,259.50,0.00),v40,z0,tPen\WObj:=wPaper;
    MoveL Offs(pOrigin,232.72,258.09,0.00),v40,z0,tPen\WObj:=wPaper;
    MoveL Offs(pOrigin,231.30,256.60,0.00),v40,z0,tPen\WObj:=wPaper;
    MoveL Offs(pOrigin,227.05,254.26,0.00),v40,fine,tPen\WObj:=wPaper;
    MoveL Offs(pOrigin,227.05,254.26,6.00),v60,z5,tPen\WObj:=wPaper;
    MoveL Offs(pOrigin,226.29,256.33,6.00),vTravel,z5,tPen\WObj:=wPaper;
    MoveL Offs(pOrigin,226.29,256.33,0.00),v60,z0,tPen\WObj:=wPaper;
    MoveL Offs(pOrigin,225.24,257.38,0.00),v40,z0,tPen\WObj:=wPaper;
    MoveL Offs(pOrigin,224.20,256.93,0.00),v40,z0,tPen\WObj:=wPaper;
    MoveL Offs(pOrigin,224.95,256.18,0.00),v40,fine,tPen\WObj:=wPaper;
    MoveL Offs(pOrigin,224.95,256.18,6.00),v60,z5,tPen\WObj:=wPaper;
    MoveL Offs(pOrigin,226.59,257.52,6.00),vTravel,z5,tPen\WObj:=wPaper;
    MoveL Offs(pOrigin,226.59,257.52,0.00),v60,z0,tPen\WObj:=wPaper;
    MoveL Offs(pOrigin,227.49,256.62,0.00),v40,fine,tPen\WObj:=wPaper;
    MoveL Offs(pOrigin,227.49,256.62,6.00),v60,z5,tPen\WObj:=wPaper;
    MoveL Offs(pOrigin,227.64,257.97,6.00),vTravel,z5,tPen\WObj:=wPaper;
    MoveL Offs(pOrigin,227.64,257.97,0.00),v60,z0,tPen\WObj:=wPaper;
    MoveL Offs(pOrigin,230.49,255.11,0.00),v40,z0,tPen\WObj:=wPaper;
    MoveL Offs(pOrigin,231.24,255.86,0.00),v40,z0,tPen\WObj:=wPaper;
    MoveL Offs(pOrigin,228.53,258.57,0.00),v40,fine,tPen\WObj:=wPaper;
    MoveL Offs(pOrigin,228.53,258.57,6.00),v60,z5,tPen\WObj:=wPaper;
    MoveL Offs(pOrigin,233.70,260.87,6.00),vTravel,z5,tPen\WObj:=wPaper;
    MoveL Offs(pOrigin,233.70,260.87,0.00),v60,z0,tPen\WObj:=wPaper;
    MoveL Offs(pOrigin,240.61,267.78,0.00),v40,z0,tPen\WObj:=wPaper;
    MoveL Offs(pOrigin,239.74,268.27,0.00),v40,z0,tPen\WObj:=wPaper;
    MoveL Offs(pOrigin,242.74,265.26,0.00),v40,fine,tPen\WObj:=wPaper;
    MoveL Offs(pOrigin,242.74,265.26,6.00),v60,z5,tPen\WObj:=wPaper;
    MoveL Offs(pOrigin,239.15,264.38,6.00),vTravel,z5,tPen\WObj:=wPaper;
    MoveL Offs(pOrigin,239.15,264.38,0.00),v60,z0,tPen\WObj:=wPaper;
    MoveL Offs(pOrigin,231.04,272.49,0.00),v40,fine,tPen\WObj:=wPaper;
    MoveL Offs(pOrigin,231.04,272.49,6.00),v60,z5,tPen\WObj:=wPaper;
    MoveL Offs(pOrigin,230.88,270.55,6.00),vTravel,z5,tPen\WObj:=wPaper;
    MoveL Offs(pOrigin,230.88,270.55,0.00),v60,z0,tPen\WObj:=wPaper;
    MoveL Offs(pOrigin,220.25,270.55,0.00),v40,fine,tPen\WObj:=wPaper;
    MoveL Offs(pOrigin,220.25,270.55,6.00),v60,z5,tPen\WObj:=wPaper;
    MoveL Offs(pOrigin,219.93,266.52,6.00),vTravel,z5,tPen\WObj:=wPaper;
    MoveL Offs(pOrigin,219.93,266.52,0.00),v60,z0,tPen\WObj:=wPaper;
    MoveL Offs(pOrigin,225.19,271.78,0.00),v40,z0,tPen\WObj:=wPaper;
    MoveL Offs(pOrigin,225.35,272.21,0.00),v40,z0,tPen\WObj:=wPaper;
    MoveL Offs(pOrigin,238.72,258.83,0.00),v40,fine,tPen\WObj:=wPaper;
    MoveL Offs(pOrigin,238.72,258.83,6.00),v60,z5,tPen\WObj:=wPaper;
    MoveL Offs(pOrigin,237.46,258.94,6.00),vTravel,z5,tPen\WObj:=wPaper;
    MoveL Offs(pOrigin,237.46,258.94,0.00),v60,z0,tPen\WObj:=wPaper;
    MoveL Offs(pOrigin,236.40,258.94,0.00),v40,fine,tPen\WObj:=wPaper;
    MoveL Offs(pOrigin,236.40,258.94,6.00),v60,z5,tPen\WObj:=wPaper;
    MoveL Offs(pOrigin,236.40,261.05,6.00),vTravel,z5,tPen\WObj:=wPaper;
    MoveL Offs(pOrigin,236.40,261.05,0.00),v60,z0,tPen\WObj:=wPaper;
    MoveL Offs(pOrigin,237.46,261.05,0.00),v40,fine,tPen\WObj:=wPaper;
    MoveL Offs(pOrigin,237.46,261.05,6.00),v60,z5,tPen\WObj:=wPaper;
    MoveL Offs(pOrigin,234.54,255.55,6.00),vTravel,z5,tPen\WObj:=wPaper;
    MoveL Offs(pOrigin,234.54,255.55,0.00),v60,z0,tPen\WObj:=wPaper;
    MoveL Offs(pOrigin,236.49,253.60,0.00),v40,z0,tPen\WObj:=wPaper;
    MoveL Offs(pOrigin,235.59,253.00,0.00),v40,z0,tPen\WObj:=wPaper;
    MoveL Offs(pOrigin,234.09,254.50,0.00),v40,z0,tPen\WObj:=wPaper;
    MoveL Offs(pOrigin,233.49,253.61,0.00),v40,z0,tPen\WObj:=wPaper;
    MoveL Offs(pOrigin,234.85,252.26,0.00),v40,z0,tPen\WObj:=wPaper;
    MoveL Offs(pOrigin,234.57,252.79,0.00),v40,z0,tPen\WObj:=wPaper;
    MoveL Offs(pOrigin,235.32,253.54,0.00),v40,fine,tPen\WObj:=wPaper;
    MoveL Offs(pOrigin,235.32,253.54,6.00),v60,z5,tPen\WObj:=wPaper;
    MoveL Offs(pOrigin,233.68,253.38,6.00),vTravel,z5,tPen\WObj:=wPaper;
    MoveL Offs(pOrigin,233.68,253.38,0.00),v60,z0,tPen\WObj:=wPaper;
    MoveL Offs(pOrigin,231.27,250.98,0.00),v40,z0,tPen\WObj:=wPaper;
    MoveL Offs(pOrigin,231.11,250.02,0.00),v40,z0,tPen\WObj:=wPaper;
    MoveL Offs(pOrigin,229.30,251.82,0.00),v40,z0,tPen\WObj:=wPaper;
    MoveL Offs(pOrigin,230.37,251.57,0.00),v40,z0,tPen\WObj:=wPaper;
    MoveL Offs(pOrigin,229.32,250.52,0.00),v40,z0,tPen\WObj:=wPaper;
    MoveL Offs(pOrigin,229.91,249.72,0.00),v40,z0,tPen\WObj:=wPaper;
    MoveL Offs(pOrigin,228.26,251.38,0.00),v40,z0,tPen\WObj:=wPaper;
  ENDPROC

  PROC DrawPart246()
    MoveL Offs(pOrigin,228.27,250.97,0.00),v40,z0,tPen\WObj:=wPaper;
    MoveL Offs(pOrigin,227.52,250.22,0.00),v40,z0,tPen\WObj:=wPaper;
    MoveL Offs(pOrigin,227.36,249.28,0.00),v40,z0,tPen\WObj:=wPaper;
    MoveL Offs(pOrigin,225.71,250.94,0.00),v40,fine,tPen\WObj:=wPaper;
    MoveL Offs(pOrigin,225.71,250.94,6.00),v60,z5,tPen\WObj:=wPaper;
    MoveL Offs(pOrigin,226.91,251.23,6.00),vTravel,z5,tPen\WObj:=wPaper;
    MoveL Offs(pOrigin,226.91,251.23,0.00),v60,z0,tPen\WObj:=wPaper;
    MoveL Offs(pOrigin,228.71,249.43,0.00),v40,fine,tPen\WObj:=wPaper;
    MoveL Offs(pOrigin,228.71,249.43,6.00),v60,z5,tPen\WObj:=wPaper;
    MoveL Offs(pOrigin,226.17,248.99,6.00),vTravel,z5,tPen\WObj:=wPaper;
    MoveL Offs(pOrigin,226.17,248.99,0.00),v60,z0,tPen\WObj:=wPaper;
    MoveL Offs(pOrigin,224.36,250.79,0.00),v40,fine,tPen\WObj:=wPaper;
    MoveL Offs(pOrigin,224.36,250.79,6.00),v60,z5,tPen\WObj:=wPaper;
    MoveL Offs(pOrigin,223.02,250.64,6.00),vTravel,z5,tPen\WObj:=wPaper;
    MoveL Offs(pOrigin,223.02,250.64,0.00),v60,z0,tPen\WObj:=wPaper;
    MoveL Offs(pOrigin,224.82,248.84,0.00),v40,fine,tPen\WObj:=wPaper;
    MoveL Offs(pOrigin,224.82,248.84,6.00),v60,z5,tPen\WObj:=wPaper;
    MoveL Offs(pOrigin,223.47,248.70,6.00),vTravel,z5,tPen\WObj:=wPaper;
    MoveL Offs(pOrigin,223.47,248.70,0.00),v60,z0,tPen\WObj:=wPaper;
    MoveL Offs(pOrigin,221.52,250.65,0.00),v40,fine,tPen\WObj:=wPaper;
    MoveL Offs(pOrigin,221.52,250.65,6.00),v60,z5,tPen\WObj:=wPaper;
    MoveL Offs(pOrigin,220.32,250.35,6.00),vTravel,z5,tPen\WObj:=wPaper;
    MoveL Offs(pOrigin,220.32,250.35,0.00),v60,z0,tPen\WObj:=wPaper;
    MoveL Offs(pOrigin,221.97,248.70,0.00),v40,fine,tPen\WObj:=wPaper;
    MoveL Offs(pOrigin,221.97,248.70,6.00),v60,z5,tPen\WObj:=wPaper;
    MoveL Offs(pOrigin,220.78,248.40,6.00),vTravel,z5,tPen\WObj:=wPaper;
    MoveL Offs(pOrigin,220.78,248.40,0.00),v60,z0,tPen\WObj:=wPaper;
    MoveL Offs(pOrigin,218.82,250.36,0.00),v40,fine,tPen\WObj:=wPaper;
    MoveL Offs(pOrigin,218.82,250.36,6.00),v60,z5,tPen\WObj:=wPaper;
    MoveL Offs(pOrigin,217.32,250.36,6.00),vTravel,z5,tPen\WObj:=wPaper;
    MoveL Offs(pOrigin,217.32,250.36,0.00),v60,z0,tPen\WObj:=wPaper;
    MoveL Offs(pOrigin,219.28,248.41,0.00),v40,fine,tPen\WObj:=wPaper;
    MoveL Offs(pOrigin,219.28,248.41,6.00),v60,z5,tPen\WObj:=wPaper;
    MoveL Offs(pOrigin,217.78,248.41,6.00),vTravel,z5,tPen\WObj:=wPaper;
    MoveL Offs(pOrigin,217.78,248.41,0.00),v60,z0,tPen\WObj:=wPaper;
    MoveL Offs(pOrigin,215.83,250.37,0.00),v40,fine,tPen\WObj:=wPaper;
    MoveL Offs(pOrigin,215.83,250.37,6.00),v60,z5,tPen\WObj:=wPaper;
    MoveL Offs(pOrigin,214.03,250.67,6.00),vTravel,z5,tPen\WObj:=wPaper;
    MoveL Offs(pOrigin,214.03,250.67,0.00),v60,z0,tPen\WObj:=wPaper;
    MoveL Offs(pOrigin,216.28,248.42,0.00),v40,fine,tPen\WObj:=wPaper;
    MoveL Offs(pOrigin,216.28,248.42,6.00),v60,z5,tPen\WObj:=wPaper;
    MoveL Offs(pOrigin,229.92,245.23,6.00),vTravel,z5,tPen\WObj:=wPaper;
    MoveL Offs(pOrigin,229.92,245.23,0.00),v60,z0,tPen\WObj:=wPaper;
    MoveL Offs(pOrigin,244.65,230.50,0.00),v40,fine,tPen\WObj:=wPaper;
    MoveL Offs(pOrigin,244.65,230.50,6.00),v60,z5,tPen\WObj:=wPaper;
    MoveL Offs(pOrigin,244.51,227.66,6.00),vTravel,z5,tPen\WObj:=wPaper;
    MoveL Offs(pOrigin,244.51,227.66,0.00),v60,z0,tPen\WObj:=wPaper;
    MoveL Offs(pOrigin,247.36,224.80,0.00),v40,z0,tPen\WObj:=wPaper;
    MoveL Offs(pOrigin,246.32,224.36,0.00),v40,z0,tPen\WObj:=wPaper;
    MoveL Offs(pOrigin,243.01,227.66,0.00),v40,fine,tPen\WObj:=wPaper;
    MoveL Offs(pOrigin,243.01,227.66,6.00),v60,z5,tPen\WObj:=wPaper;
    MoveL Offs(pOrigin,242.86,226.32,6.00),vTravel,z5,tPen\WObj:=wPaper;
    MoveL Offs(pOrigin,242.86,226.32,0.00),v60,z0,tPen\WObj:=wPaper;
    MoveL Offs(pOrigin,241.66,227.52,0.00),v40,z0,tPen\WObj:=wPaper;
    MoveL Offs(pOrigin,241.22,226.47,0.00),v40,z0,tPen\WObj:=wPaper;
    MoveL Offs(pOrigin,240.46,227.22,0.00),v40,fine,tPen\WObj:=wPaper;
    MoveL Offs(pOrigin,240.46,227.22,6.00),v60,z5,tPen\WObj:=wPaper;
    MoveL Offs(pOrigin,240.31,230.37,6.00),vTravel,z5,tPen\WObj:=wPaper;
    MoveL Offs(pOrigin,240.31,230.37,0.00),v60,z0,tPen\WObj:=wPaper;
    MoveL Offs(pOrigin,231.59,239.08,0.00),v40,z0,tPen\WObj:=wPaper;
    MoveL Offs(pOrigin,230.78,238.54,0.00),v40,z0,tPen\WObj:=wPaper;
    MoveL Offs(pOrigin,222.67,230.43,0.00),v40,z0,tPen\WObj:=wPaper;
    MoveL Offs(pOrigin,222.18,230.57,0.00),v40,z0,tPen\WObj:=wPaper;
    MoveL Offs(pOrigin,227.29,225.46,0.00),v40,fine,tPen\WObj:=wPaper;
    MoveL Offs(pOrigin,227.29,225.46,6.00),v60,z5,tPen\WObj:=wPaper;
    MoveL Offs(pOrigin,226.10,226.40,6.00),vTravel,z5,tPen\WObj:=wPaper;
    MoveL Offs(pOrigin,226.10,226.40,0.00),v60,z0,tPen\WObj:=wPaper;
    MoveL Offs(pOrigin,240.68,240.97,0.00),v40,fine,tPen\WObj:=wPaper;
    MoveL Offs(pOrigin,240.68,240.97,6.00),v60,z5,tPen\WObj:=wPaper;
    MoveL Offs(pOrigin,239.73,239.81,6.00),vTravel,z5,tPen\WObj:=wPaper;
    MoveL Offs(pOrigin,239.73,239.81,0.00),v60,z0,tPen\WObj:=wPaper;
    MoveL Offs(pOrigin,239.73,234.71,0.00),v40,z0,tPen\WObj:=wPaper;
    MoveL Offs(pOrigin,240.44,234.29,0.00),v40,z0,tPen\WObj:=wPaper;
    MoveL Offs(pOrigin,241.71,233.86,0.00),v40,z0,tPen\WObj:=wPaper;
    MoveL Offs(pOrigin,242.77,234.50,0.00),v40,z0,tPen\WObj:=wPaper;
    MoveL Offs(pOrigin,243.41,234.65,0.00),v40,z0,tPen\WObj:=wPaper;
    MoveL Offs(pOrigin,224.29,234.65,0.00),v40,z0,tPen\WObj:=wPaper;
    MoveL Offs(pOrigin,224.94,234.29,0.00),v40,z0,tPen\WObj:=wPaper;
    MoveL Offs(pOrigin,224.94,228.34,0.00),v40,fine,tPen\WObj:=wPaper;
    MoveL Offs(pOrigin,224.94,228.34,6.00),v60,z5,tPen\WObj:=wPaper;
    MoveL Offs(pOrigin,226.00,227.70,6.00),vTravel,z5,tPen\WObj:=wPaper;
    MoveL Offs(pOrigin,226.00,227.70,0.00),v60,z0,tPen\WObj:=wPaper;
    MoveL Offs(pOrigin,226.00,234.71,0.00),v40,z0,tPen\WObj:=wPaper;
    MoveL Offs(pOrigin,225.77,235.35,0.00),v40,z0,tPen\WObj:=wPaper;
    MoveL Offs(pOrigin,224.71,235.77,0.00),v40,z0,tPen\WObj:=wPaper;
    MoveL Offs(pOrigin,225.77,235.35,0.00),v40,z0,tPen\WObj:=wPaper;
    MoveL Offs(pOrigin,226.62,235.99,0.00),v40,z0,tPen\WObj:=wPaper;
    MoveL Offs(pOrigin,227.26,235.99,0.00),v40,z0,tPen\WObj:=wPaper;
    MoveL Offs(pOrigin,227.26,235.99,0.00),v40,z0,tPen\WObj:=wPaper;
    MoveL Offs(pOrigin,227.69,235.21,0.00),v40,z0,tPen\WObj:=wPaper;
    MoveL Offs(pOrigin,228.11,235.14,0.00),v40,z0,tPen\WObj:=wPaper;
    MoveL Offs(pOrigin,228.68,235.42,0.00),v40,z0,tPen\WObj:=wPaper;
    MoveL Offs(pOrigin,228.96,236.20,0.00),v40,z0,tPen\WObj:=wPaper;
    MoveL Offs(pOrigin,229.17,235.56,0.00),v40,z0,tPen\WObj:=wPaper;
    MoveL Offs(pOrigin,229.17,229.40,0.00),v40,fine,tPen\WObj:=wPaper;
    MoveL Offs(pOrigin,229.17,229.40,6.00),v60,z5,tPen\WObj:=wPaper;
    MoveL Offs(pOrigin,230.22,230.04,6.00),vTravel,z5,tPen\WObj:=wPaper;
    MoveL Offs(pOrigin,230.22,230.04,0.00),v60,z0,tPen\WObj:=wPaper;
    MoveL Offs(pOrigin,230.22,235.78,0.00),v40,fine,tPen\WObj:=wPaper;
    MoveL Offs(pOrigin,230.22,235.78,6.00),v60,z5,tPen\WObj:=wPaper;
    MoveL Offs(pOrigin,231.28,236.62,6.00),vTravel,z5,tPen\WObj:=wPaper;
    MoveL Offs(pOrigin,231.28,236.62,0.00),v60,z0,tPen\WObj:=wPaper;
    MoveL Offs(pOrigin,231.28,230.46,0.00),v40,z0,tPen\WObj:=wPaper;
    MoveL Offs(pOrigin,230.38,230.75,0.00),v40,z0,tPen\WObj:=wPaper;
    MoveL Offs(pOrigin,229.67,230.68,0.00),v40,z0,tPen\WObj:=wPaper;
    MoveL Offs(pOrigin,229.88,231.67,0.00),v40,z0,tPen\WObj:=wPaper;
    MoveL Offs(pOrigin,230.59,231.31,0.00),v40,z0,tPen\WObj:=wPaper;
    MoveL Offs(pOrigin,230.38,230.75,0.00),v40,z0,tPen\WObj:=wPaper;
    MoveL Offs(pOrigin,230.66,231.31,0.00),v40,z0,tPen\WObj:=wPaper;
    MoveL Offs(pOrigin,231.51,231.31,0.00),v40,z0,tPen\WObj:=wPaper;
    MoveL Offs(pOrigin,232.36,231.95,0.00),v40,z0,tPen\WObj:=wPaper;
    MoveL Offs(pOrigin,232.33,232.38,0.00),v40,z0,tPen\WObj:=wPaper;
    MoveL Offs(pOrigin,232.33,237.26,0.00),v40,z0,tPen\WObj:=wPaper;
    MoveL Offs(pOrigin,232.15,237.05,0.00),v40,z0,tPen\WObj:=wPaper;
    MoveL Offs(pOrigin,232.57,237.26,0.00),v40,z0,tPen\WObj:=wPaper;
    MoveL Offs(pOrigin,232.57,238.11,0.00),v40,z0,tPen\WObj:=wPaper;
    MoveL Offs(pOrigin,233.39,237.69,0.00),v40,z0,tPen\WObj:=wPaper;
    MoveL Offs(pOrigin,233.39,233.01,0.00),v40,z0,tPen\WObj:=wPaper;
    MoveL Offs(pOrigin,234.06,232.16,0.00),v40,z0,tPen\WObj:=wPaper;
    MoveL Offs(pOrigin,234.49,231.60,0.00),v40,z0,tPen\WObj:=wPaper;
  ENDPROC

  PROC DrawPart247()
    MoveL Offs(pOrigin,235.98,232.59,0.00),v40,z0,tPen\WObj:=wPaper;
    MoveL Offs(pOrigin,235.76,232.16,0.00),v40,z0,tPen\WObj:=wPaper;
    MoveL Offs(pOrigin,235.98,232.59,0.00),v40,z0,tPen\WObj:=wPaper;
    MoveL Offs(pOrigin,235.76,232.16,0.00),v40,z0,tPen\WObj:=wPaper;
    MoveL Offs(pOrigin,235.12,232.54,0.00),v40,z0,tPen\WObj:=wPaper;
    MoveL Offs(pOrigin,223.44,232.54,0.00),v40,z0,tPen\WObj:=wPaper;
    MoveL Offs(pOrigin,223.89,233.01,0.00),v40,z0,tPen\WObj:=wPaper;
    MoveL Offs(pOrigin,223.89,229.40,0.00),v40,z0,tPen\WObj:=wPaper;
    MoveL Offs(pOrigin,223.65,229.37,0.00),v40,z0,tPen\WObj:=wPaper;
    MoveL Offs(pOrigin,230.66,229.37,0.00),v40,fine,tPen\WObj:=wPaper;
    MoveL Offs(pOrigin,230.66,229.37,6.00),v60,z5,tPen\WObj:=wPaper;
    MoveL Offs(pOrigin,230.73,228.00,6.00),vTravel,z5,tPen\WObj:=wPaper;
    MoveL Offs(pOrigin,230.73,228.00,0.00),v60,z0,tPen\WObj:=wPaper;
    MoveL Offs(pOrigin,223.21,235.51,0.00),v40,z0,tPen\WObj:=wPaper;
    MoveL Offs(pOrigin,222.47,234.77,0.00),v40,z0,tPen\WObj:=wPaper;
    MoveL Offs(pOrigin,229.83,227.40,0.00),v40,z0,tPen\WObj:=wPaper;
    MoveL Offs(pOrigin,229.23,226.51,0.00),v40,z0,tPen\WObj:=wPaper;
    MoveL Offs(pOrigin,222.17,233.57,0.00),v40,fine,tPen\WObj:=wPaper;
    MoveL Offs(pOrigin,222.17,233.57,6.00),v60,z5,tPen\WObj:=wPaper;
    MoveL Offs(pOrigin,223.65,233.59,6.00),vTravel,z5,tPen\WObj:=wPaper;
    MoveL Offs(pOrigin,223.65,233.59,0.00),v60,z0,tPen\WObj:=wPaper;
    MoveL Offs(pOrigin,238.52,233.59,0.00),v40,z0,tPen\WObj:=wPaper;
    MoveL Offs(pOrigin,238.67,234.50,0.00),v40,z0,tPen\WObj:=wPaper;
    MoveL Offs(pOrigin,238.67,239.81,0.00),v40,z0,tPen\WObj:=wPaper;
    MoveL Offs(pOrigin,238.95,240.45,0.00),v40,z0,tPen\WObj:=wPaper;
    MoveL Offs(pOrigin,239.80,239.39,0.00),v40,z0,tPen\WObj:=wPaper;
    MoveL Offs(pOrigin,240.37,239.46,0.00),v40,z0,tPen\WObj:=wPaper;
    MoveL Offs(pOrigin,241.07,240.17,0.00),v40,z0,tPen\WObj:=wPaper;
    MoveL Offs(pOrigin,241.71,239.95,0.00),v40,z0,tPen\WObj:=wPaper;
    MoveL Offs(pOrigin,242.14,239.18,0.00),v40,z0,tPen\WObj:=wPaper;
    MoveL Offs(pOrigin,242.14,239.18,0.00),v40,z0,tPen\WObj:=wPaper;
    MoveL Offs(pOrigin,243.62,239.18,0.00),v40,z0,tPen\WObj:=wPaper;
    MoveL Offs(pOrigin,243.62,239.18,0.00),v40,z0,tPen\WObj:=wPaper;
    MoveL Offs(pOrigin,244.48,239.60,0.00),v40,z0,tPen\WObj:=wPaper;
    MoveL Offs(pOrigin,245.75,239.60,0.00),v40,z0,tPen\WObj:=wPaper;
    MoveL Offs(pOrigin,245.11,238.87,0.00),v40,z0,tPen\WObj:=wPaper;
    MoveL Offs(pOrigin,268.91,238.87,0.00),v40,z0,tPen\WObj:=wPaper;
    MoveL Offs(pOrigin,268.24,238.54,0.00),v40,z0,tPen\WObj:=wPaper;
    MoveL Offs(pOrigin,268.24,233.01,0.00),v40,fine,tPen\WObj:=wPaper;
    MoveL Offs(pOrigin,268.24,233.01,6.00),v60,z5,tPen\WObj:=wPaper;
    MoveL Offs(pOrigin,266.13,233.22,6.00),vTravel,z5,tPen\WObj:=wPaper;
    MoveL Offs(pOrigin,266.13,233.22,0.00),v60,z0,tPen\WObj:=wPaper;
    MoveL Offs(pOrigin,266.13,239.60,0.00),v40,z0,tPen\WObj:=wPaper;
    MoveL Offs(pOrigin,265.07,239.81,0.00),v40,z0,tPen\WObj:=wPaper;
    MoveL Offs(pOrigin,265.07,233.86,0.00),v40,z0,tPen\WObj:=wPaper;
    MoveL Offs(pOrigin,264.01,234.29,0.00),v40,z0,tPen\WObj:=wPaper;
    MoveL Offs(pOrigin,264.01,239.81,0.00),v40,z0,tPen\WObj:=wPaper;
    MoveL Offs(pOrigin,262.96,239.81,0.00),v40,z0,tPen\WObj:=wPaper;
    MoveL Offs(pOrigin,262.96,234.29,0.00),v40,z0,tPen\WObj:=wPaper;
    MoveL Offs(pOrigin,261.90,234.29,0.00),v40,z0,tPen\WObj:=wPaper;
    MoveL Offs(pOrigin,261.90,239.81,0.00),v40,z0,tPen\WObj:=wPaper;
    MoveL Offs(pOrigin,260.85,239.81,0.00),v40,z0,tPen\WObj:=wPaper;
    MoveL Offs(pOrigin,260.85,235.78,0.00),v40,z0,tPen\WObj:=wPaper;
    MoveL Offs(pOrigin,260.41,234.93,0.00),v40,z0,tPen\WObj:=wPaper;
    MoveL Offs(pOrigin,261.26,234.50,0.00),v40,z0,tPen\WObj:=wPaper;
    MoveL Offs(pOrigin,263.17,235.28,0.00),v40,z0,tPen\WObj:=wPaper;
    MoveL Offs(pOrigin,264.02,235.07,0.00),v40,z0,tPen\WObj:=wPaper;
    MoveL Offs(pOrigin,264.24,234.71,0.00),v40,fine,tPen\WObj:=wPaper;
    MoveL Offs(pOrigin,264.24,234.71,6.00),v60,z5,tPen\WObj:=wPaper;
    MoveL Offs(pOrigin,264.17,233.10,6.00),vTravel,z5,tPen\WObj:=wPaper;
    MoveL Offs(pOrigin,264.17,233.10,0.00),v60,z0,tPen\WObj:=wPaper;
    MoveL Offs(pOrigin,269.73,238.66,0.00),v40,z0,tPen\WObj:=wPaper;
    MoveL Offs(pOrigin,270.39,239.11,0.00),v40,z0,tPen\WObj:=wPaper;
    MoveL Offs(pOrigin,266.33,243.17,0.00),v40,fine,tPen\WObj:=wPaper;
    MoveL Offs(pOrigin,266.33,243.17,6.00),v60,z5,tPen\WObj:=wPaper;
    MoveL Offs(pOrigin,266.74,241.65,6.00),vTravel,z5,tPen\WObj:=wPaper;
    MoveL Offs(pOrigin,266.74,241.65,0.00),v60,z0,tPen\WObj:=wPaper;
    MoveL Offs(pOrigin,257.88,232.78,0.00),v40,fine,tPen\WObj:=wPaper;
    MoveL Offs(pOrigin,257.88,232.78,6.00),v60,z5,tPen\WObj:=wPaper;
    MoveL Offs(pOrigin,259.14,233.23,6.00),vTravel,z5,tPen\WObj:=wPaper;
    MoveL Offs(pOrigin,259.14,233.23,0.00),v60,z0,tPen\WObj:=wPaper;
    MoveL Offs(pOrigin,259.42,234.71,0.00),v40,z0,tPen\WObj:=wPaper;
    MoveL Offs(pOrigin,260.41,234.93,0.00),v40,fine,tPen\WObj:=wPaper;
    MoveL Offs(pOrigin,260.41,234.93,6.00),v60,z5,tPen\WObj:=wPaper;
    MoveL Offs(pOrigin,261.69,234.93,6.00),vTravel,z5,tPen\WObj:=wPaper;
    MoveL Offs(pOrigin,261.69,234.93,0.00),v60,z0,tPen\WObj:=wPaper;
    MoveL Offs(pOrigin,261.48,235.42,0.00),v40,z0,tPen\WObj:=wPaper;
    MoveL Offs(pOrigin,260.48,235.56,0.00),v40,z0,tPen\WObj:=wPaper;
    MoveL Offs(pOrigin,259.56,236.98,0.00),v40,z0,tPen\WObj:=wPaper;
    MoveL Offs(pOrigin,258.71,237.26,0.00),v40,fine,tPen\WObj:=wPaper;
    MoveL Offs(pOrigin,258.71,237.26,6.00),v60,z5,tPen\WObj:=wPaper;
    MoveL Offs(pOrigin,259.79,236.20,6.00),vTravel,z5,tPen\WObj:=wPaper;
    MoveL Offs(pOrigin,259.79,236.20,0.00),v60,z0,tPen\WObj:=wPaper;
    MoveL Offs(pOrigin,259.79,240.02,0.00),v40,fine,tPen\WObj:=wPaper;
    MoveL Offs(pOrigin,259.79,240.02,6.00),v60,z5,tPen\WObj:=wPaper;
    MoveL Offs(pOrigin,260.84,240.88,6.00),vTravel,z5,tPen\WObj:=wPaper;
    MoveL Offs(pOrigin,260.84,240.88,0.00),v60,z0,tPen\WObj:=wPaper;
    MoveL Offs(pOrigin,258.29,241.73,0.00),v40,z0,tPen\WObj:=wPaper;
    MoveL Offs(pOrigin,254.89,241.94,0.00),v40,z0,tPen\WObj:=wPaper;
    MoveL Offs(pOrigin,254.89,241.94,0.00),v40,z0,tPen\WObj:=wPaper;
    MoveL Offs(pOrigin,254.32,242.36,0.00),v40,z0,tPen\WObj:=wPaper;
    MoveL Offs(pOrigin,254.18,243.64,0.00),v40,z0,tPen\WObj:=wPaper;
    MoveL Offs(pOrigin,255.74,244.91,0.00),v40,z0,tPen\WObj:=wPaper;
    MoveL Offs(pOrigin,256.16,245.76,0.00),v40,z0,tPen\WObj:=wPaper;
    MoveL Offs(pOrigin,256.16,248.52,0.00),v40,z0,tPen\WObj:=wPaper;
    MoveL Offs(pOrigin,255.74,250.23,0.00),v40,fine,tPen\WObj:=wPaper;
    MoveL Offs(pOrigin,255.74,250.23,6.00),v60,z5,tPen\WObj:=wPaper;
    MoveL Offs(pOrigin,254.78,248.75,6.00),vTravel,z5,tPen\WObj:=wPaper;
    MoveL Offs(pOrigin,254.78,248.75,0.00),v60,z0,tPen\WObj:=wPaper;
    MoveL Offs(pOrigin,257.18,246.34,0.00),v40,z0,tPen\WObj:=wPaper;
    MoveL Offs(pOrigin,256.74,245.30,0.00),v40,z0,tPen\WObj:=wPaper;
    MoveL Offs(pOrigin,255.23,246.80,0.00),v40,z0,tPen\WObj:=wPaper;
    MoveL Offs(pOrigin,254.79,245.75,0.00),v40,z0,tPen\WObj:=wPaper;
    MoveL Offs(pOrigin,256.44,244.10,0.00),v40,fine,tPen\WObj:=wPaper;
    MoveL Offs(pOrigin,256.44,244.10,6.00),v60,z5,tPen\WObj:=wPaper;
    MoveL Offs(pOrigin,255.74,245.12,6.00),vTravel,z5,tPen\WObj:=wPaper;
    MoveL Offs(pOrigin,255.74,245.12,0.00),v60,z0,tPen\WObj:=wPaper;
    MoveL Offs(pOrigin,255.95,245.55,0.00),v40,z0,tPen\WObj:=wPaper;
    MoveL Offs(pOrigin,255.74,245.12,0.00),v40,fine,tPen\WObj:=wPaper;
    MoveL Offs(pOrigin,255.74,245.12,6.00),v60,z5,tPen\WObj:=wPaper;
    MoveL Offs(pOrigin,253.27,244.60,6.00),vTravel,z5,tPen\WObj:=wPaper;
    MoveL Offs(pOrigin,253.27,244.60,0.00),v60,z0,tPen\WObj:=wPaper;
    MoveL Offs(pOrigin,242.15,233.49,0.00),v40,fine,tPen\WObj:=wPaper;
    MoveL Offs(pOrigin,242.15,233.49,6.00),v60,z5,tPen\WObj:=wPaper;
    MoveL Offs(pOrigin,241.84,235.14,6.00),vTravel,z5,tPen\WObj:=wPaper;
    MoveL Offs(pOrigin,241.84,235.14,0.00),v60,z0,tPen\WObj:=wPaper;
    MoveL Offs(pOrigin,241.84,238.96,0.00),v40,z0,tPen\WObj:=wPaper;
    MoveL Offs(pOrigin,240.78,239.39,0.00),v40,z0,tPen\WObj:=wPaper;
    MoveL Offs(pOrigin,240.78,234.92,0.00),v40,fine,tPen\WObj:=wPaper;
    MoveL Offs(pOrigin,240.78,234.92,6.00),v60,z5,tPen\WObj:=wPaper;
  ENDPROC

  PROC DrawPart248()
    MoveL Offs(pOrigin,242.77,235.77,6.00),vTravel,z5,tPen\WObj:=wPaper;
    MoveL Offs(pOrigin,242.77,235.77,0.00),v60,z0,tPen\WObj:=wPaper;
    MoveL Offs(pOrigin,242.77,234.93,0.00),v40,z0,tPen\WObj:=wPaper;
    MoveL Offs(pOrigin,243.20,234.50,0.00),v40,z0,tPen\WObj:=wPaper;
    MoveL Offs(pOrigin,244.69,235.56,0.00),v40,z0,tPen\WObj:=wPaper;
    MoveL Offs(pOrigin,245.11,236.41,0.00),v40,z0,tPen\WObj:=wPaper;
    MoveL Offs(pOrigin,244.90,238.11,0.00),v40,z0,tPen\WObj:=wPaper;
    MoveL Offs(pOrigin,244.90,238.11,0.00),v40,z0,tPen\WObj:=wPaper;
    MoveL Offs(pOrigin,244.48,238.11,0.00),v40,z0,tPen\WObj:=wPaper;
    MoveL Offs(pOrigin,243.62,239.18,0.00),v40,z0,tPen\WObj:=wPaper;
    MoveL Offs(pOrigin,243.84,238.87,0.00),v40,z0,tPen\WObj:=wPaper;
    MoveL Offs(pOrigin,234.06,238.87,0.00),v40,z0,tPen\WObj:=wPaper;
    MoveL Offs(pOrigin,234.45,238.11,0.00),v40,z0,tPen\WObj:=wPaper;
    MoveL Offs(pOrigin,234.45,233.44,0.00),v40,z0,tPen\WObj:=wPaper;
    MoveL Offs(pOrigin,235.50,233.65,0.00),v40,z0,tPen\WObj:=wPaper;
    MoveL Offs(pOrigin,235.50,238.75,0.00),v40,fine,tPen\WObj:=wPaper;
    MoveL Offs(pOrigin,235.50,238.75,6.00),v60,z5,tPen\WObj:=wPaper;
    MoveL Offs(pOrigin,236.56,239.39,6.00),vTravel,z5,tPen\WObj:=wPaper;
    MoveL Offs(pOrigin,236.56,239.39,0.00),v60,z0,tPen\WObj:=wPaper;
    MoveL Offs(pOrigin,236.56,234.08,0.00),v40,fine,tPen\WObj:=wPaper;
    MoveL Offs(pOrigin,236.56,234.08,6.00),v60,z5,tPen\WObj:=wPaper;
    MoveL Offs(pOrigin,237.46,232.80,6.00),vTravel,z5,tPen\WObj:=wPaper;
    MoveL Offs(pOrigin,237.46,232.80,0.00),v60,z0,tPen\WObj:=wPaper;
    MoveL Offs(pOrigin,237.68,233.23,0.00),v40,z0,tPen\WObj:=wPaper;
    MoveL Offs(pOrigin,237.46,232.80,0.00),v40,fine,tPen\WObj:=wPaper;
    MoveL Offs(pOrigin,237.46,232.80,6.00),v60,z5,tPen\WObj:=wPaper;
    MoveL Offs(pOrigin,237.80,230.63,6.00),vTravel,z5,tPen\WObj:=wPaper;
    MoveL Offs(pOrigin,237.80,230.63,0.00),v60,z0,tPen\WObj:=wPaper;
    MoveL Offs(pOrigin,251.92,244.75,0.00),v40,z0,tPen\WObj:=wPaper;
    MoveL Offs(pOrigin,252.34,244.49,0.00),v40,z0,tPen\WObj:=wPaper;
    MoveL Offs(pOrigin,253.75,243.85,0.00),v40,z0,tPen\WObj:=wPaper;
    MoveL Offs(pOrigin,253.54,243.21,0.00),v40,z0,tPen\WObj:=wPaper;
    MoveL Offs(pOrigin,252.76,242.57,0.00),v40,fine,tPen\WObj:=wPaper;
    MoveL Offs(pOrigin,252.76,242.57,6.00),v60,z5,tPen\WObj:=wPaper;
    MoveL Offs(pOrigin,252.24,245.31,6.00),vTravel,z5,tPen\WObj:=wPaper;
    MoveL Offs(pOrigin,252.24,245.31,0.00),v60,z0,tPen\WObj:=wPaper;
    MoveL Offs(pOrigin,266.97,230.59,0.00),v40,fine,tPen\WObj:=wPaper;
    MoveL Offs(pOrigin,266.97,230.59,6.00),v60,z5,tPen\WObj:=wPaper;
    MoveL Offs(pOrigin,263.97,232.09,6.00),vTravel,z5,tPen\WObj:=wPaper;
    MoveL Offs(pOrigin,263.97,232.09,0.00),v60,z0,tPen\WObj:=wPaper;
    MoveL Offs(pOrigin,250.90,245.17,0.00),v40,fine,tPen\WObj:=wPaper;
    MoveL Offs(pOrigin,250.90,245.17,6.00),v60,z5,tPen\WObj:=wPaper;
    MoveL Offs(pOrigin,249.70,244.87,6.00),vTravel,z5,tPen\WObj:=wPaper;
    MoveL Offs(pOrigin,249.70,244.87,0.00),v60,z0,tPen\WObj:=wPaper;
    MoveL Offs(pOrigin,262.17,232.40,0.00),v40,z0,tPen\WObj:=wPaper;
    MoveL Offs(pOrigin,262.67,233.10,0.00),v40,z0,tPen\WObj:=wPaper;
    MoveL Offs(pOrigin,269.29,239.71,0.00),v40,z0,tPen\WObj:=wPaper;
    MoveL Offs(pOrigin,268.69,240.61,0.00),v40,z0,tPen\WObj:=wPaper;
    MoveL Offs(pOrigin,260.73,232.64,0.00),v40,z0,tPen\WObj:=wPaper;
    MoveL Offs(pOrigin,261.12,231.95,0.00),v40,z0,tPen\WObj:=wPaper;
    MoveL Offs(pOrigin,248.65,244.42,0.00),v40,z0,tPen\WObj:=wPaper;
    MoveL Offs(pOrigin,247.90,243.68,0.00),v40,z0,tPen\WObj:=wPaper;
    MoveL Offs(pOrigin,260.08,231.51,0.00),v40,fine,tPen\WObj:=wPaper;
    MoveL Offs(pOrigin,260.08,231.51,6.00),v60,z5,tPen\WObj:=wPaper;
    MoveL Offs(pOrigin,258.88,231.21,6.00),vTravel,z5,tPen\WObj:=wPaper;
    MoveL Offs(pOrigin,258.88,231.21,0.00),v60,z0,tPen\WObj:=wPaper;
    MoveL Offs(pOrigin,247.16,242.93,0.00),v40,fine,tPen\WObj:=wPaper;
    MoveL Offs(pOrigin,247.16,242.93,6.00),v60,z5,tPen\WObj:=wPaper;
    MoveL Offs(pOrigin,242.89,238.32,6.00),vTravel,z5,tPen\WObj:=wPaper;
    MoveL Offs(pOrigin,242.89,238.32,0.00),v60,z0,tPen\WObj:=wPaper;
    MoveL Offs(pOrigin,242.89,235.56,0.00),v40,z0,tPen\WObj:=wPaper;
    MoveL Offs(pOrigin,243.95,235.99,0.00),v40,z0,tPen\WObj:=wPaper;
    MoveL Offs(pOrigin,243.95,237.26,0.00),v40,fine,tPen\WObj:=wPaper;
    MoveL Offs(pOrigin,243.95,237.26,6.00),v60,z5,tPen\WObj:=wPaper;
    MoveL Offs(pOrigin,244.90,235.56,6.00),vTravel,z5,tPen\WObj:=wPaper;
    MoveL Offs(pOrigin,244.90,235.56,0.00),v60,z0,tPen\WObj:=wPaper;
    MoveL Offs(pOrigin,245.11,235.99,0.00),v40,z0,tPen\WObj:=wPaper;
    MoveL Offs(pOrigin,244.90,235.56,0.00),v40,fine,tPen\WObj:=wPaper;
    MoveL Offs(pOrigin,244.90,235.56,6.00),v60,z5,tPen\WObj:=wPaper;
    MoveL Offs(pOrigin,240.95,232.28,6.00),vTravel,z5,tPen\WObj:=wPaper;
    MoveL Offs(pOrigin,240.95,232.28,0.00),v60,z0,tPen\WObj:=wPaper;
    MoveL Offs(pOrigin,239.60,230.93,0.00),v40,z0,tPen\WObj:=wPaper;
    MoveL Offs(pOrigin,239.11,230.07,0.00),v40,z0,tPen\WObj:=wPaper;
    MoveL Offs(pOrigin,230.54,238.64,0.00),v40,z0,tPen\WObj:=wPaper;
    MoveL Offs(pOrigin,231.09,237.90,0.00),v40,z0,tPen\WObj:=wPaper;
    MoveL Offs(pOrigin,232.15,237.05,0.00),v40,fine,tPen\WObj:=wPaper;
    MoveL Offs(pOrigin,232.15,237.05,6.00),v60,z5,tPen\WObj:=wPaper;
    MoveL Offs(pOrigin,232.64,239.53,6.00),vTravel,z5,tPen\WObj:=wPaper;
    MoveL Offs(pOrigin,232.64,239.53,0.00),v60,z0,tPen\WObj:=wPaper;
    MoveL Offs(pOrigin,241.65,230.51,0.00),v40,fine,tPen\WObj:=wPaper;
    MoveL Offs(pOrigin,241.65,230.51,6.00),v60,z5,tPen\WObj:=wPaper;
    MoveL Offs(pOrigin,237.76,229.93,6.00),vTravel,z5,tPen\WObj:=wPaper;
    MoveL Offs(pOrigin,237.76,229.93,0.00),v60,z0,tPen\WObj:=wPaper;
    MoveL Offs(pOrigin,229.35,238.34,0.00),v40,fine,tPen\WObj:=wPaper;
    MoveL Offs(pOrigin,229.35,238.34,6.00),v60,z5,tPen\WObj:=wPaper;
    MoveL Offs(pOrigin,228.23,237.49,6.00),vTravel,z5,tPen\WObj:=wPaper;
    MoveL Offs(pOrigin,228.23,237.49,0.00),v60,z0,tPen\WObj:=wPaper;
    MoveL Offs(pOrigin,222.67,231.93,0.00),v40,fine,tPen\WObj:=wPaper;
    MoveL Offs(pOrigin,222.67,231.93,6.00),v60,z5,tPen\WObj:=wPaper;
    MoveL Offs(pOrigin,223.12,229.38,6.00),vTravel,z5,tPen\WObj:=wPaper;
    MoveL Offs(pOrigin,223.12,229.38,0.00),v60,z0,tPen\WObj:=wPaper;
    MoveL Offs(pOrigin,233.33,239.60,0.00),v40,fine,tPen\WObj:=wPaper;
    MoveL Offs(pOrigin,233.33,239.60,6.00),v60,z5,tPen\WObj:=wPaper;
    MoveL Offs(pOrigin,227.05,235.14,6.00),vTravel,z5,tPen\WObj:=wPaper;
    MoveL Offs(pOrigin,227.05,235.14,0.00),v60,z0,tPen\WObj:=wPaper;
    MoveL Offs(pOrigin,227.05,227.70,0.00),v40,z0,tPen\WObj:=wPaper;
    MoveL Offs(pOrigin,227.90,227.26,0.00),v40,z0,tPen\WObj:=wPaper;
    MoveL Offs(pOrigin,225.56,227.26,0.00),v40,fine,tPen\WObj:=wPaper;
    MoveL Offs(pOrigin,225.56,227.26,6.00),v60,z5,tPen\WObj:=wPaper;
    MoveL Offs(pOrigin,219.61,224.30,6.00),vTravel,z5,tPen\WObj:=wPaper;
    MoveL Offs(pOrigin,219.61,224.30,0.00),v60,z0,tPen\WObj:=wPaper;
    MoveL Offs(pOrigin,221.95,220.48,0.00),v40,z0,tPen\WObj:=wPaper;
    MoveL Offs(pOrigin,223.23,218.99,0.00),v40,fine,tPen\WObj:=wPaper;
    MoveL Offs(pOrigin,223.23,218.99,6.00),v60,z5,tPen\WObj:=wPaper;
    MoveL Offs(pOrigin,209.84,222.39,6.00),vTravel,z5,tPen\WObj:=wPaper;
    MoveL Offs(pOrigin,209.84,222.39,0.00),v60,z0,tPen\WObj:=wPaper;
    MoveL Offs(pOrigin,209.62,222.81,0.00),v40,z0,tPen\WObj:=wPaper;
    MoveL Offs(pOrigin,209.84,222.39,0.00),v40,fine,tPen\WObj:=wPaper;
    MoveL Offs(pOrigin,209.84,222.39,6.00),v60,z5,tPen\WObj:=wPaper;
    MoveL Offs(pOrigin,212.27,208.36,6.00),vTravel,z5,tPen\WObj:=wPaper;
    MoveL Offs(pOrigin,212.27,208.36,0.00),v60,z0,tPen\WObj:=wPaper;
    MoveL Offs(pOrigin,212.27,207.30,0.00),v40,z0,tPen\WObj:=wPaper;
    MoveL Offs(pOrigin,212.81,206.88,0.00),v40,z0,tPen\WObj:=wPaper;
    MoveL Offs(pOrigin,213.02,207.30,0.00),v40,z0,tPen\WObj:=wPaper;
    MoveL Offs(pOrigin,212.81,206.88,0.00),v40,fine,tPen\WObj:=wPaper;
    MoveL Offs(pOrigin,212.81,206.88,6.00),v60,z5,tPen\WObj:=wPaper;
    MoveL Offs(pOrigin,230.10,188.31,6.00),vTravel,z5,tPen\WObj:=wPaper;
    MoveL Offs(pOrigin,230.10,188.31,0.00),v60,z0,tPen\WObj:=wPaper;
    MoveL Offs(pOrigin,232.20,186.20,0.00),v40,z0,tPen\WObj:=wPaper;
    MoveL Offs(pOrigin,231.72,187.13,0.00),v40,z0,tPen\WObj:=wPaper;
  ENDPROC

  PROC DrawPart249()
    MoveL Offs(pOrigin,230.45,187.13,0.00),v40,z0,tPen\WObj:=wPaper;
    MoveL Offs(pOrigin,230.88,186.69,0.00),v40,z0,tPen\WObj:=wPaper;
    MoveL Offs(pOrigin,231.30,187.11,0.00),v40,z0,tPen\WObj:=wPaper;
    MoveL Offs(pOrigin,230.88,186.69,0.00),v40,z0,tPen\WObj:=wPaper;
    MoveL Offs(pOrigin,230.66,186.07,0.00),v40,z0,tPen\WObj:=wPaper;
    MoveL Offs(pOrigin,229.60,186.07,0.00),v40,z0,tPen\WObj:=wPaper;
    MoveL Offs(pOrigin,229.18,185.02,0.00),v40,z0,tPen\WObj:=wPaper;
    MoveL Offs(pOrigin,230.24,185.02,0.00),v40,fine,tPen\WObj:=wPaper;
    MoveL Offs(pOrigin,230.24,185.02,6.00),v60,z5,tPen\WObj:=wPaper;
    MoveL Offs(pOrigin,231.30,185.61,6.00),vTravel,z5,tPen\WObj:=wPaper;
    MoveL Offs(pOrigin,231.30,185.61,0.00),v60,z0,tPen\WObj:=wPaper;
    MoveL Offs(pOrigin,229.35,187.56,0.00),v40,fine,tPen\WObj:=wPaper;
    MoveL Offs(pOrigin,229.35,187.56,6.00),v60,z5,tPen\WObj:=wPaper;
    MoveL Offs(pOrigin,226.27,165.25,6.00),vTravel,z5,tPen\WObj:=wPaper;
    MoveL Offs(pOrigin,226.27,165.25,0.00),v60,z0,tPen\WObj:=wPaper;
    MoveL Offs(pOrigin,234.24,157.28,0.00),v40,fine,tPen\WObj:=wPaper;
    MoveL Offs(pOrigin,234.24,157.28,6.00),v60,z5,tPen\WObj:=wPaper;
    MoveL Offs(pOrigin,233.64,156.09,6.00),vTravel,z5,tPen\WObj:=wPaper;
    MoveL Offs(pOrigin,233.64,156.09,0.00),v60,z0,tPen\WObj:=wPaper;
    MoveL Offs(pOrigin,233.43,156.51,0.00),v40,z0,tPen\WObj:=wPaper;
    MoveL Offs(pOrigin,233.64,156.09,0.00),v40,fine,tPen\WObj:=wPaper;
    MoveL Offs(pOrigin,233.64,156.09,6.00),v60,z5,tPen\WObj:=wPaper;
    MoveL Offs(pOrigin,231.99,156.54,6.00),vTravel,z5,tPen\WObj:=wPaper;
    MoveL Offs(pOrigin,231.99,156.54,0.00),v60,z0,tPen\WObj:=wPaper;
    MoveL Offs(pOrigin,236.35,152.18,0.00),v40,fine,tPen\WObj:=wPaper;
    MoveL Offs(pOrigin,236.35,152.18,6.00),v60,z5,tPen\WObj:=wPaper;
    MoveL Offs(pOrigin,234.56,150.99,6.00),vTravel,z5,tPen\WObj:=wPaper;
    MoveL Offs(pOrigin,234.56,150.99,0.00),v60,z0,tPen\WObj:=wPaper;
    MoveL Offs(pOrigin,238.01,147.54,0.00),v40,fine,tPen\WObj:=wPaper;
    MoveL Offs(pOrigin,238.01,147.54,6.00),v60,z5,tPen\WObj:=wPaper;
    MoveL Offs(pOrigin,231.72,147.85,6.00),vTravel,z5,tPen\WObj:=wPaper;
    MoveL Offs(pOrigin,231.72,147.85,0.00),v60,z0,tPen\WObj:=wPaper;
    MoveL Offs(pOrigin,227.96,151.61,0.00),v40,z0,tPen\WObj:=wPaper;
    MoveL Offs(pOrigin,228.42,152.55,0.00),v40,z0,tPen\WObj:=wPaper;
    MoveL Offs(pOrigin,230.38,154.50,0.00),v40,z0,tPen\WObj:=wPaper;
    MoveL Offs(pOrigin,230.80,154.75,0.00),v40,z0,tPen\WObj:=wPaper;
    MoveL Offs(pOrigin,227.04,158.50,0.00),v40,fine,tPen\WObj:=wPaper;
    MoveL Offs(pOrigin,227.04,158.50,6.00),v60,z5,tPen\WObj:=wPaper;
    MoveL Offs(pOrigin,226.89,160.15,6.00),vTravel,z5,tPen\WObj:=wPaper;
    MoveL Offs(pOrigin,226.89,160.15,0.00),v60,z0,tPen\WObj:=wPaper;
    MoveL Offs(pOrigin,230.80,156.25,0.00),v40,z0,tPen\WObj:=wPaper;
    MoveL Offs(pOrigin,230.23,155.85,0.00),v40,z0,tPen\WObj:=wPaper;
    MoveL Offs(pOrigin,228.28,153.90,0.00),v40,z0,tPen\WObj:=wPaper;
    MoveL Offs(pOrigin,228.75,154.39,0.00),v40,z0,tPen\WObj:=wPaper;
    MoveL Offs(pOrigin,229.81,154.39,0.00),v40,z0,tPen\WObj:=wPaper;
    MoveL Offs(pOrigin,229.81,155.45,0.00),v40,z0,tPen\WObj:=wPaper;
    MoveL Offs(pOrigin,228.75,155.45,0.00),v40,z0,tPen\WObj:=wPaper;
    MoveL Offs(pOrigin,227.98,155.10,0.00),v40,z0,tPen\WObj:=wPaper;
    MoveL Offs(pOrigin,230.23,157.35,0.00),v40,z0,tPen\WObj:=wPaper;
    MoveL Offs(pOrigin,229.60,157.56,0.00),v40,z0,tPen\WObj:=wPaper;
    MoveL Offs(pOrigin,228.54,157.56,0.00),v40,z0,tPen\WObj:=wPaper;
    MoveL Offs(pOrigin,228.54,156.50,0.00),v40,z0,tPen\WObj:=wPaper;
    MoveL Offs(pOrigin,229.60,156.50,0.00),v40,fine,tPen\WObj:=wPaper;
    MoveL Offs(pOrigin,229.60,156.50,6.00),v60,z5,tPen\WObj:=wPaper;
    MoveL Offs(pOrigin,230.64,157.89,6.00),vTravel,z5,tPen\WObj:=wPaper;
    MoveL Offs(pOrigin,230.64,157.89,0.00),v60,z0,tPen\WObj:=wPaper;
    MoveL Offs(pOrigin,226.73,161.80,0.00),v40,z0,tPen\WObj:=wPaper;
    MoveL Offs(pOrigin,227.90,161.78,0.00),v40,z0,tPen\WObj:=wPaper;
    MoveL Offs(pOrigin,229.18,161.78,0.00),v40,z0,tPen\WObj:=wPaper;
    MoveL Offs(pOrigin,229.18,160.73,0.00),v40,z0,tPen\WObj:=wPaper;
    MoveL Offs(pOrigin,228.11,160.73,0.00),v40,z0,tPen\WObj:=wPaper;
    MoveL Offs(pOrigin,227.55,160.64,0.00),v40,z0,tPen\WObj:=wPaper;
    MoveL Offs(pOrigin,231.00,164.09,0.00),v40,fine,tPen\WObj:=wPaper;
    MoveL Offs(pOrigin,231.00,164.09,6.00),v60,z5,tPen\WObj:=wPaper;
    MoveL Offs(pOrigin,227.50,155.06,6.00),vTravel,z5,tPen\WObj:=wPaper;
    MoveL Offs(pOrigin,227.50,155.06,0.00),v60,z0,tPen\WObj:=wPaper;
    MoveL Offs(pOrigin,231.26,151.30,0.00),v40,z0,tPen\WObj:=wPaper;
    MoveL Offs(pOrigin,230.81,150.46,0.00),v40,z0,tPen\WObj:=wPaper;
    MoveL Offs(pOrigin,228.86,148.51,0.00),v40,z0,tPen\WObj:=wPaper;
    MoveL Offs(pOrigin,228.27,148.31,0.00),v40,z0,tPen\WObj:=wPaper;
    MoveL Offs(pOrigin,231.88,144.71,0.00),v40,z0,tPen\WObj:=wPaper;
    MoveL Offs(pOrigin,231.40,145.07,0.00),v40,z0,tPen\WObj:=wPaper;
    MoveL Offs(pOrigin,229.29,142.97,0.00),v40,z0,tPen\WObj:=wPaper;
    MoveL Offs(pOrigin,228.89,143.22,0.00),v40,z0,tPen\WObj:=wPaper;
    MoveL Offs(pOrigin,232.49,139.61,0.00),v40,z0,tPen\WObj:=wPaper;
    MoveL Offs(pOrigin,231.83,139.53,0.00),v40,z0,tPen\WObj:=wPaper;
    MoveL Offs(pOrigin,229.87,137.58,0.00),v40,z0,tPen\WObj:=wPaper;
    MoveL Offs(pOrigin,230.45,137.50,0.00),v40,z0,tPen\WObj:=wPaper;
    MoveL Offs(pOrigin,231.51,137.50,0.00),v40,z0,tPen\WObj:=wPaper;
    MoveL Offs(pOrigin,232.12,136.83,0.00),v40,z0,tPen\WObj:=wPaper;
    MoveL Offs(pOrigin,230.17,134.88,0.00),v40,z0,tPen\WObj:=wPaper;
    MoveL Offs(pOrigin,229.51,135.13,0.00),v40,z0,tPen\WObj:=wPaper;
    MoveL Offs(pOrigin,233.12,131.52,0.00),v40,z0,tPen\WObj:=wPaper;
    MoveL Offs(pOrigin,232.55,131.29,0.00),v40,z0,tPen\WObj:=wPaper;
    MoveL Offs(pOrigin,230.60,129.34,0.00),v40,z0,tPen\WObj:=wPaper;
    MoveL Offs(pOrigin,231.09,129.05,0.00),v40,z0,tPen\WObj:=wPaper;
    MoveL Offs(pOrigin,232.15,129.05,0.00),v40,z0,tPen\WObj:=wPaper;
    MoveL Offs(pOrigin,232.84,128.60,0.00),v40,z0,tPen\WObj:=wPaper;
    MoveL Offs(pOrigin,230.59,126.34,0.00),v40,z0,tPen\WObj:=wPaper;
    MoveL Offs(pOrigin,230.14,127.04,0.00),v40,z0,tPen\WObj:=wPaper;
    MoveL Offs(pOrigin,233.59,123.58,0.00),v40,z0,tPen\WObj:=wPaper;
    MoveL Offs(pOrigin,233.12,122.91,0.00),v40,z0,tPen\WObj:=wPaper;
    MoveL Offs(pOrigin,231.02,120.80,0.00),v40,z0,tPen\WObj:=wPaper;
    MoveL Offs(pOrigin,231.51,120.60,0.00),v40,z0,tPen\WObj:=wPaper;
    MoveL Offs(pOrigin,232.58,120.60,0.00),v40,z0,tPen\WObj:=wPaper;
    MoveL Offs(pOrigin,233.60,120.59,0.00),v40,z0,tPen\WObj:=wPaper;
    MoveL Offs(pOrigin,230.45,123.74,0.00),v40,fine,tPen\WObj:=wPaper;
    MoveL Offs(pOrigin,230.45,123.74,6.00),v60,z5,tPen\WObj:=wPaper;
    MoveL Offs(pOrigin,231.30,124.82,6.00),vTravel,z5,tPen\WObj:=wPaper;
    MoveL Offs(pOrigin,231.30,124.82,0.00),v60,z0,tPen\WObj:=wPaper;
    MoveL Offs(pOrigin,232.36,124.82,0.00),v40,z0,tPen\WObj:=wPaper;
    MoveL Offs(pOrigin,233.44,125.23,0.00),v40,z0,tPen\WObj:=wPaper;
    MoveL Offs(pOrigin,229.98,128.69,0.00),v40,z0,tPen\WObj:=wPaper;
    MoveL Offs(pOrigin,230.59,127.84,0.00),v40,z0,tPen\WObj:=wPaper;
    MoveL Offs(pOrigin,232.85,130.10,0.00),v40,z0,tPen\WObj:=wPaper;
    MoveL Offs(pOrigin,233.12,130.02,0.00),v40,z0,tPen\WObj:=wPaper;
    MoveL Offs(pOrigin,229.67,133.48,0.00),v40,z0,tPen\WObj:=wPaper;
    MoveL Offs(pOrigin,230.16,133.38,0.00),v40,z0,tPen\WObj:=wPaper;
    MoveL Offs(pOrigin,232.41,135.64,0.00),v40,z0,tPen\WObj:=wPaper;
    MoveL Offs(pOrigin,231.72,135.38,0.00),v40,z0,tPen\WObj:=wPaper;
    MoveL Offs(pOrigin,230.66,135.38,0.00),v40,z0,tPen\WObj:=wPaper;
    MoveL Offs(pOrigin,230.66,136.44,0.00),v40,z0,tPen\WObj:=wPaper;
    MoveL Offs(pOrigin,231.72,136.44,0.00),v40,z0,tPen\WObj:=wPaper;
    MoveL Offs(pOrigin,232.80,136.32,0.00),v40,z0,tPen\WObj:=wPaper;
    MoveL Offs(pOrigin,229.05,140.07,0.00),v40,z0,tPen\WObj:=wPaper;
    MoveL Offs(pOrigin,229.58,140.27,0.00),v40,z0,tPen\WObj:=wPaper;
    MoveL Offs(pOrigin,231.69,142.38,0.00),v40,z0,tPen\WObj:=wPaper;
    MoveL Offs(pOrigin,231.09,142.78,0.00),v40,z0,tPen\WObj:=wPaper;
    MoveL Offs(pOrigin,230.02,142.78,0.00),v40,fine,tPen\WObj:=wPaper;
    MoveL Offs(pOrigin,230.02,142.78,6.00),v60,z5,tPen\WObj:=wPaper;
  ENDPROC

  PROC DrawPart250()
    MoveL Offs(pOrigin,232.03,143.06,6.00),vTravel,z5,tPen\WObj:=wPaper;
    MoveL Offs(pOrigin,232.03,143.06,0.00),v60,z0,tPen\WObj:=wPaper;
    MoveL Offs(pOrigin,228.43,146.67,0.00),v40,z0,tPen\WObj:=wPaper;
    MoveL Offs(pOrigin,229.00,147.16,0.00),v40,z0,tPen\WObj:=wPaper;
    MoveL Offs(pOrigin,230.96,149.11,0.00),v40,z0,tPen\WObj:=wPaper;
    MoveL Offs(pOrigin,230.45,149.11,0.00),v40,z0,tPen\WObj:=wPaper;
    MoveL Offs(pOrigin,229.39,149.11,0.00),v40,z0,tPen\WObj:=wPaper;
    MoveL Offs(pOrigin,229.18,150.17,0.00),v40,z0,tPen\WObj:=wPaper;
    MoveL Offs(pOrigin,230.24,150.17,0.00),v40,fine,tPen\WObj:=wPaper;
    MoveL Offs(pOrigin,230.24,150.17,6.00),v60,z5,tPen\WObj:=wPaper;
    MoveL Offs(pOrigin,231.42,149.65,6.00),vTravel,z5,tPen\WObj:=wPaper;
    MoveL Offs(pOrigin,231.42,149.65,0.00),v60,z0,tPen\WObj:=wPaper;
    MoveL Offs(pOrigin,227.81,153.26,0.00),v40,z0,tPen\WObj:=wPaper;
    MoveL Offs(pOrigin,228.96,153.34,0.00),v40,z0,tPen\WObj:=wPaper;
    MoveL Offs(pOrigin,230.02,153.34,0.00),v40,fine,tPen\WObj:=wPaper;
    MoveL Offs(pOrigin,230.02,153.34,6.00),v60,z5,tPen\WObj:=wPaper;
    MoveL Offs(pOrigin,230.95,147.62,6.00),vTravel,z5,tPen\WObj:=wPaper;
    MoveL Offs(pOrigin,230.95,147.62,0.00),v60,z0,tPen\WObj:=wPaper;
    MoveL Offs(pOrigin,229.00,145.66,0.00),v40,z0,tPen\WObj:=wPaper;
    MoveL Offs(pOrigin,228.58,145.02,0.00),v40,z0,tPen\WObj:=wPaper;
    MoveL Offs(pOrigin,232.34,141.26,0.00),v40,z0,tPen\WObj:=wPaper;
    MoveL Offs(pOrigin,231.83,141.03,0.00),v40,z0,tPen\WObj:=wPaper;
    MoveL Offs(pOrigin,229.58,138.77,0.00),v40,z0,tPen\WObj:=wPaper;
    MoveL Offs(pOrigin,229.35,138.27,0.00),v40,z0,tPen\WObj:=wPaper;
    MoveL Offs(pOrigin,232.96,134.67,0.00),v40,z0,tPen\WObj:=wPaper;
    MoveL Offs(pOrigin,232.41,134.14,0.00),v40,z0,tPen\WObj:=wPaper;
    MoveL Offs(pOrigin,230.46,132.19,0.00),v40,z0,tPen\WObj:=wPaper;
    MoveL Offs(pOrigin,230.88,132.22,0.00),v40,z0,tPen\WObj:=wPaper;
    MoveL Offs(pOrigin,231.94,132.22,0.00),v40,z0,tPen\WObj:=wPaper;
    MoveL Offs(pOrigin,231.94,133.27,0.00),v40,z0,tPen\WObj:=wPaper;
    MoveL Offs(pOrigin,230.88,133.27,0.00),v40,z0,tPen\WObj:=wPaper;
    MoveL Offs(pOrigin,230.88,134.33,0.00),v40,z0,tPen\WObj:=wPaper;
    MoveL Offs(pOrigin,231.94,134.33,0.00),v40,fine,tPen\WObj:=wPaper;
    MoveL Offs(pOrigin,231.94,134.33,6.00),v60,z5,tPen\WObj:=wPaper;
    MoveL Offs(pOrigin,232.15,131.16,6.00),vTravel,z5,tPen\WObj:=wPaper;
    MoveL Offs(pOrigin,232.15,131.16,0.00),v60,z0,tPen\WObj:=wPaper;
    MoveL Offs(pOrigin,231.09,131.16,0.00),v40,z0,tPen\WObj:=wPaper;
    MoveL Offs(pOrigin,231.09,130.10,0.00),v40,z0,tPen\WObj:=wPaper;
    MoveL Offs(pOrigin,232.15,130.10,0.00),v40,fine,tPen\WObj:=wPaper;
    MoveL Offs(pOrigin,232.15,130.10,6.00),v60,z5,tPen\WObj:=wPaper;
    MoveL Offs(pOrigin,232.36,127.99,6.00),vTravel,z5,tPen\WObj:=wPaper;
    MoveL Offs(pOrigin,232.36,127.99,0.00),v60,z0,tPen\WObj:=wPaper;
    MoveL Offs(pOrigin,231.30,127.99,0.00),v40,z0,tPen\WObj:=wPaper;
    MoveL Offs(pOrigin,231.30,126.94,0.00),v40,z0,tPen\WObj:=wPaper;
    MoveL Offs(pOrigin,232.36,126.94,0.00),v40,fine,tPen\WObj:=wPaper;
    MoveL Offs(pOrigin,232.36,126.94,6.00),v60,z5,tPen\WObj:=wPaper;
    MoveL Offs(pOrigin,233.43,128.23,6.00),vTravel,z5,tPen\WObj:=wPaper;
    MoveL Offs(pOrigin,233.43,128.23,0.00),v60,z0,tPen\WObj:=wPaper;
    MoveL Offs(pOrigin,229.67,131.98,0.00),v40,fine,tPen\WObj:=wPaper;
    MoveL Offs(pOrigin,229.67,131.98,6.00),v60,z5,tPen\WObj:=wPaper;
    MoveL Offs(pOrigin,235.21,133.91,6.00),vTravel,z5,tPen\WObj:=wPaper;
    MoveL Offs(pOrigin,235.21,133.91,0.00),v60,z0,tPen\WObj:=wPaper;
    MoveL Offs(pOrigin,236.86,132.26,0.00),v40,fine,tPen\WObj:=wPaper;
    MoveL Offs(pOrigin,236.86,132.26,6.00),v60,z5,tPen\WObj:=wPaper;
    MoveL Offs(pOrigin,235.66,131.96,6.00),vTravel,z5,tPen\WObj:=wPaper;
    MoveL Offs(pOrigin,235.66,131.96,0.00),v60,z0,tPen\WObj:=wPaper;
    MoveL Offs(pOrigin,237.17,130.46,0.00),v40,z0,tPen\WObj:=wPaper;
    MoveL Offs(pOrigin,236.12,130.02,0.00),v40,z0,tPen\WObj:=wPaper;
    MoveL Offs(pOrigin,237.62,128.51,0.00),v40,z0,tPen\WObj:=wPaper;
    MoveL Offs(pOrigin,236.57,128.07,0.00),v40,z0,tPen\WObj:=wPaper;
    MoveL Offs(pOrigin,237.93,126.71,0.00),v40,z0,tPen\WObj:=wPaper;
    MoveL Offs(pOrigin,237.18,125.97,0.00),v40,z0,tPen\WObj:=wPaper;
    MoveL Offs(pOrigin,237.93,125.22,0.00),v40,fine,tPen\WObj:=wPaper;
    MoveL Offs(pOrigin,237.93,125.22,6.00),v60,z5,tPen\WObj:=wPaper;
    MoveL Offs(pOrigin,238.31,121.88,6.00),vTravel,z5,tPen\WObj:=wPaper;
    MoveL Offs(pOrigin,238.31,121.88,0.00),v60,z0,tPen\WObj:=wPaper;
    MoveL Offs(pOrigin,237.04,129.10,0.00),v40,z0,tPen\WObj:=wPaper;
    MoveL Offs(pOrigin,233.85,142.06,0.00),v40,fine,tPen\WObj:=wPaper;
    MoveL Offs(pOrigin,233.85,142.06,6.00),v60,z5,tPen\WObj:=wPaper;
    MoveL Offs(pOrigin,231.30,140.66,6.00),vTravel,z5,tPen\WObj:=wPaper;
    MoveL Offs(pOrigin,231.30,140.66,0.00),v60,z0,tPen\WObj:=wPaper;
    MoveL Offs(pOrigin,230.24,140.66,0.00),v40,fine,tPen\WObj:=wPaper;
    MoveL Offs(pOrigin,230.24,140.66,6.00),v60,z5,tPen\WObj:=wPaper;
    MoveL Offs(pOrigin,230.45,138.55,6.00),vTravel,z5,tPen\WObj:=wPaper;
    MoveL Offs(pOrigin,230.45,138.55,0.00),v60,z0,tPen\WObj:=wPaper;
    MoveL Offs(pOrigin,231.51,138.55,0.00),v40,fine,tPen\WObj:=wPaper;
    MoveL Offs(pOrigin,231.51,138.55,6.00),v60,z5,tPen\WObj:=wPaper;
    MoveL Offs(pOrigin,234.60,137.51,6.00),vTravel,z5,tPen\WObj:=wPaper;
    MoveL Offs(pOrigin,234.60,137.51,0.00),v60,z0,tPen\WObj:=wPaper;
    MoveL Offs(pOrigin,235.65,136.46,0.00),v40,z0,tPen\WObj:=wPaper;
    MoveL Offs(pOrigin,234.75,135.86,0.00),v40,z0,tPen\WObj:=wPaper;
    MoveL Offs(pOrigin,236.41,134.21,0.00),v40,fine,tPen\WObj:=wPaper;
    MoveL Offs(pOrigin,236.41,134.21,6.00),v60,z5,tPen\WObj:=wPaper;
    MoveL Offs(pOrigin,230.14,125.54,6.00),vTravel,z5,tPen\WObj:=wPaper;
    MoveL Offs(pOrigin,230.14,125.54,0.00),v60,z0,tPen\WObj:=wPaper;
    MoveL Offs(pOrigin,233.60,122.08,0.00),v40,z0,tPen\WObj:=wPaper;
    MoveL Offs(pOrigin,232.58,122.71,0.00),v40,z0,tPen\WObj:=wPaper;
    MoveL Offs(pOrigin,231.51,122.71,0.00),v40,z0,tPen\WObj:=wPaper;
    MoveL Offs(pOrigin,230.45,122.24,0.00),v40,z0,tPen\WObj:=wPaper;
    MoveL Offs(pOrigin,233.61,119.09,0.00),v40,z0,tPen\WObj:=wPaper;
    MoveL Offs(pOrigin,233.11,118.41,0.00),v40,z0,tPen\WObj:=wPaper;
    MoveL Offs(pOrigin,231.01,116.31,0.00),v40,z0,tPen\WObj:=wPaper;
    MoveL Offs(pOrigin,230.47,116.25,0.00),v40,z0,tPen\WObj:=wPaper;
    MoveL Offs(pOrigin,233.77,112.95,0.00),v40,z0,tPen\WObj:=wPaper;
    MoveL Offs(pOrigin,232.79,113.21,0.00),v40,z0,tPen\WObj:=wPaper;
    MoveL Offs(pOrigin,231.72,113.21,0.00),v40,z0,tPen\WObj:=wPaper;
    MoveL Offs(pOrigin,231.00,113.31,0.00),v40,z0,tPen\WObj:=wPaper;
    MoveL Offs(pOrigin,233.10,115.42,0.00),v40,z0,tPen\WObj:=wPaper;
    MoveL Offs(pOrigin,232.79,115.32,0.00),v40,z0,tPen\WObj:=wPaper;
    MoveL Offs(pOrigin,231.72,115.32,0.00),v40,z0,tPen\WObj:=wPaper;
    MoveL Offs(pOrigin,231.00,114.81,0.00),v40,z0,tPen\WObj:=wPaper;
    MoveL Offs(pOrigin,233.11,116.91,0.00),v40,z0,tPen\WObj:=wPaper;
    MoveL Offs(pOrigin,232.79,117.43,0.00),v40,z0,tPen\WObj:=wPaper;
    MoveL Offs(pOrigin,231.72,117.43,0.00),v40,z0,tPen\WObj:=wPaper;
    MoveL Offs(pOrigin,231.72,116.38,0.00),v40,z0,tPen\WObj:=wPaper;
    MoveL Offs(pOrigin,232.79,116.38,0.00),v40,fine,tPen\WObj:=wPaper;
    MoveL Offs(pOrigin,232.79,116.38,6.00),v60,z5,tPen\WObj:=wPaper;
    MoveL Offs(pOrigin,233.92,115.79,6.00),vTravel,z5,tPen\WObj:=wPaper;
    MoveL Offs(pOrigin,233.92,115.79,0.00),v60,z0,tPen\WObj:=wPaper;
    MoveL Offs(pOrigin,230.46,119.25,0.00),v40,fine,tPen\WObj:=wPaper;
    MoveL Offs(pOrigin,230.46,119.25,6.00),v60,z5,tPen\WObj:=wPaper;
    MoveL Offs(pOrigin,230.46,120.75,6.00),vTravel,z5,tPen\WObj:=wPaper;
    MoveL Offs(pOrigin,230.46,120.75,0.00),v60,z0,tPen\WObj:=wPaper;
    MoveL Offs(pOrigin,233.91,117.29,0.00),v40,fine,tPen\WObj:=wPaper;
    MoveL Offs(pOrigin,233.91,117.29,6.00),v60,z5,tPen\WObj:=wPaper;
    MoveL Offs(pOrigin,232.79,114.26,6.00),vTravel,z5,tPen\WObj:=wPaper;
    MoveL Offs(pOrigin,232.79,114.26,0.00),v60,z0,tPen\WObj:=wPaper;
    MoveL Offs(pOrigin,231.72,114.26,0.00),v40,fine,tPen\WObj:=wPaper;
    MoveL Offs(pOrigin,231.72,114.26,6.00),v60,z5,tPen\WObj:=wPaper;
    MoveL Offs(pOrigin,230.47,114.75,6.00),vTravel,z5,tPen\WObj:=wPaper;
  ENDPROC

  PROC DrawPart251()
    MoveL Offs(pOrigin,230.47,114.75,0.00),v60,z0,tPen\WObj:=wPaper;
    MoveL Offs(pOrigin,233.78,111.45,0.00),v40,z0,tPen\WObj:=wPaper;
    MoveL Offs(pOrigin,233.09,110.92,0.00),v40,z0,tPen\WObj:=wPaper;
    MoveL Offs(pOrigin,230.98,108.82,0.00),v40,z0,tPen\WObj:=wPaper;
    MoveL Offs(pOrigin,230.49,108.76,0.00),v40,z0,tPen\WObj:=wPaper;
    MoveL Offs(pOrigin,233.50,105.76,0.00),v40,z0,tPen\WObj:=wPaper;
    MoveL Offs(pOrigin,232.58,105.82,0.00),v40,z0,tPen\WObj:=wPaper;
    MoveL Offs(pOrigin,231.51,105.82,0.00),v40,z0,tPen\WObj:=wPaper;
    MoveL Offs(pOrigin,230.83,105.67,0.00),v40,z0,tPen\WObj:=wPaper;
    MoveL Offs(pOrigin,233.08,107.93,0.00),v40,z0,tPen\WObj:=wPaper;
    MoveL Offs(pOrigin,232.58,107.93,0.00),v40,z0,tPen\WObj:=wPaper;
    MoveL Offs(pOrigin,231.51,107.93,0.00),v40,fine,tPen\WObj:=wPaper;
    MoveL Offs(pOrigin,231.51,107.93,6.00),v60,z5,tPen\WObj:=wPaper;
    MoveL Offs(pOrigin,230.35,107.41,6.00),vTravel,z5,tPen\WObj:=wPaper;
    MoveL Offs(pOrigin,230.35,107.41,0.00),v60,z0,tPen\WObj:=wPaper;
    MoveL Offs(pOrigin,233.50,104.26,0.00),v40,z0,tPen\WObj:=wPaper;
    MoveL Offs(pOrigin,232.58,103.70,0.00),v40,z0,tPen\WObj:=wPaper;
    MoveL Offs(pOrigin,231.30,103.70,0.00),v40,z0,tPen\WObj:=wPaper;
    MoveL Offs(pOrigin,231.30,102.65,0.00),v40,z0,tPen\WObj:=wPaper;
    MoveL Offs(pOrigin,232.36,102.65,0.00),v40,z0,tPen\WObj:=wPaper;
    MoveL Offs(pOrigin,232.91,103.28,0.00),v40,z0,tPen\WObj:=wPaper;
    MoveL Offs(pOrigin,230.51,100.88,0.00),v40,z0,tPen\WObj:=wPaper;
    MoveL Offs(pOrigin,230.07,100.22,0.00),v40,z0,tPen\WObj:=wPaper;
    MoveL Offs(pOrigin,232.92,97.37,0.00),v40,z0,tPen\WObj:=wPaper;
    MoveL Offs(pOrigin,232.45,96.84,0.00),v40,z0,tPen\WObj:=wPaper;
    MoveL Offs(pOrigin,229.89,94.28,0.00),v40,z0,tPen\WObj:=wPaper;
    MoveL Offs(pOrigin,229.49,94.83,0.00),v40,z0,tPen\WObj:=wPaper;
    MoveL Offs(pOrigin,232.49,91.83,0.00),v40,fine,tPen\WObj:=wPaper;
    MoveL Offs(pOrigin,232.49,91.83,6.00),v60,z5,tPen\WObj:=wPaper;
    MoveL Offs(pOrigin,232.79,93.03,6.00),vTravel,z5,tPen\WObj:=wPaper;
    MoveL Offs(pOrigin,232.79,93.03,0.00),v60,z0,tPen\WObj:=wPaper;
    MoveL Offs(pOrigin,229.63,96.18,0.00),v40,fine,tPen\WObj:=wPaper;
    MoveL Offs(pOrigin,229.63,96.18,6.00),v60,z5,tPen\WObj:=wPaper;
    MoveL Offs(pOrigin,229.93,97.38,6.00),vTravel,z5,tPen\WObj:=wPaper;
    MoveL Offs(pOrigin,229.93,97.38,0.00),v60,z0,tPen\WObj:=wPaper;
    MoveL Offs(pOrigin,232.78,94.52,0.00),v40,z0,tPen\WObj:=wPaper;
    MoveL Offs(pOrigin,231.72,94.20,0.00),v40,z0,tPen\WObj:=wPaper;
    MoveL Offs(pOrigin,230.66,94.20,0.00),v40,fine,tPen\WObj:=wPaper;
    MoveL Offs(pOrigin,230.66,94.20,6.00),v60,z5,tPen\WObj:=wPaper;
    MoveL Offs(pOrigin,230.88,96.31,6.00),vTravel,z5,tPen\WObj:=wPaper;
    MoveL Offs(pOrigin,230.88,96.31,0.00),v60,z0,tPen\WObj:=wPaper;
    MoveL Offs(pOrigin,231.94,96.31,0.00),v40,z0,tPen\WObj:=wPaper;
    MoveL Offs(pOrigin,231.94,97.37,0.00),v40,z0,tPen\WObj:=wPaper;
    MoveL Offs(pOrigin,230.88,97.37,0.00),v40,z0,tPen\WObj:=wPaper;
    MoveL Offs(pOrigin,230.35,97.73,0.00),v40,z0,tPen\WObj:=wPaper;
    MoveL Offs(pOrigin,232.76,100.14,0.00),v40,z0,tPen\WObj:=wPaper;
    MoveL Offs(pOrigin,233.06,100.21,0.00),v40,z0,tPen\WObj:=wPaper;
    MoveL Offs(pOrigin,230.06,103.22,0.00),v40,fine,tPen\WObj:=wPaper;
    MoveL Offs(pOrigin,230.06,103.22,6.00),v60,z5,tPen\WObj:=wPaper;
    MoveL Offs(pOrigin,230.36,104.42,6.00),vTravel,z5,tPen\WObj:=wPaper;
    MoveL Offs(pOrigin,230.36,104.42,0.00),v60,z0,tPen\WObj:=wPaper;
    MoveL Offs(pOrigin,233.36,101.41,0.00),v40,z0,tPen\WObj:=wPaper;
    MoveL Offs(pOrigin,232.91,101.78,0.00),v40,z0,tPen\WObj:=wPaper;
    MoveL Offs(pOrigin,230.36,99.23,0.00),v40,z0,tPen\WObj:=wPaper;
    MoveL Offs(pOrigin,229.92,98.88,0.00),v40,z0,tPen\WObj:=wPaper;
    MoveL Offs(pOrigin,232.93,95.87,0.00),v40,fine,tPen\WObj:=wPaper;
    MoveL Offs(pOrigin,232.93,95.87,6.00),v60,z5,tPen\WObj:=wPaper;
    MoveL Offs(pOrigin,232.15,98.42,6.00),vTravel,z5,tPen\WObj:=wPaper;
    MoveL Offs(pOrigin,232.15,98.42,0.00),v60,z0,tPen\WObj:=wPaper;
    MoveL Offs(pOrigin,231.09,98.42,0.00),v40,z0,tPen\WObj:=wPaper;
    MoveL Offs(pOrigin,231.09,99.48,0.00),v40,z0,tPen\WObj:=wPaper;
    MoveL Offs(pOrigin,232.15,99.48,0.00),v40,z0,tPen\WObj:=wPaper;
    MoveL Offs(pOrigin,232.36,100.54,0.00),v40,z0,tPen\WObj:=wPaper;
    MoveL Offs(pOrigin,231.30,100.54,0.00),v40,z0,tPen\WObj:=wPaper;
    MoveL Offs(pOrigin,231.30,101.59,0.00),v40,z0,tPen\WObj:=wPaper;
    MoveL Offs(pOrigin,232.36,101.59,0.00),v40,fine,tPen\WObj:=wPaper;
    MoveL Offs(pOrigin,232.36,101.59,6.00),v60,z5,tPen\WObj:=wPaper;
    MoveL Offs(pOrigin,233.36,102.91,6.00),vTravel,z5,tPen\WObj:=wPaper;
    MoveL Offs(pOrigin,233.36,102.91,0.00),v60,z0,tPen\WObj:=wPaper;
    MoveL Offs(pOrigin,230.35,105.92,0.00),v40,fine,tPen\WObj:=wPaper;
    MoveL Offs(pOrigin,230.35,105.92,6.00),v60,z5,tPen\WObj:=wPaper;
    MoveL Offs(pOrigin,233.49,107.25,6.00),vTravel,z5,tPen\WObj:=wPaper;
    MoveL Offs(pOrigin,233.49,107.25,0.00),v60,z0,tPen\WObj:=wPaper;
    MoveL Offs(pOrigin,230.49,110.26,0.00),v40,fine,tPen\WObj:=wPaper;
    MoveL Offs(pOrigin,230.49,110.26,6.00),v60,z5,tPen\WObj:=wPaper;
    MoveL Offs(pOrigin,231.72,111.10,6.00),vTravel,z5,tPen\WObj:=wPaper;
    MoveL Offs(pOrigin,231.72,111.10,0.00),v60,z0,tPen\WObj:=wPaper;
    MoveL Offs(pOrigin,232.79,111.10,0.00),v40,z0,tPen\WObj:=wPaper;
    MoveL Offs(pOrigin,233.48,110.25,0.00),v40,z0,tPen\WObj:=wPaper;
    MoveL Offs(pOrigin,230.48,113.26,0.00),v40,fine,tPen\WObj:=wPaper;
    MoveL Offs(pOrigin,230.48,113.26,6.00),v60,z5,tPen\WObj:=wPaper;
    MoveL Offs(pOrigin,230.48,111.76,6.00),vTravel,z5,tPen\WObj:=wPaper;
    MoveL Offs(pOrigin,230.48,111.76,0.00),v60,z0,tPen\WObj:=wPaper;
    MoveL Offs(pOrigin,233.49,108.75,0.00),v40,fine,tPen\WObj:=wPaper;
    MoveL Offs(pOrigin,233.49,108.75,6.00),v60,z5,tPen\WObj:=wPaper;
    MoveL Offs(pOrigin,247.41,112.75,6.00),vTravel,z5,tPen\WObj:=wPaper;
    MoveL Offs(pOrigin,247.41,112.75,0.00),v60,z0,tPen\WObj:=wPaper;
    MoveL Offs(pOrigin,250.71,109.45,0.00),v40,z0,tPen\WObj:=wPaper;
    MoveL Offs(pOrigin,250.43,110.40,0.00),v40,z0,tPen\WObj:=wPaper;
    MoveL Offs(pOrigin,249.36,110.82,0.00),v40,z0,tPen\WObj:=wPaper;
    MoveL Offs(pOrigin,248.65,111.68,0.00),v40,z0,tPen\WObj:=wPaper;
    MoveL Offs(pOrigin,248.30,113.80,0.00),v40,z0,tPen\WObj:=wPaper;
    MoveL Offs(pOrigin,249.36,115.50,0.00),v40,z0,tPen\WObj:=wPaper;
    MoveL Offs(pOrigin,251.49,116.14,0.00),v40,z0,tPen\WObj:=wPaper;
    MoveL Offs(pOrigin,253.19,115.29,0.00),v40,z0,tPen\WObj:=wPaper;
    MoveL Offs(pOrigin,253.75,114.44,0.00),v40,z0,tPen\WObj:=wPaper;
    MoveL Offs(pOrigin,254.04,112.74,0.00),v40,z0,tPen\WObj:=wPaper;
    MoveL Offs(pOrigin,253.75,111.89,0.00),v40,z0,tPen\WObj:=wPaper;
    MoveL Offs(pOrigin,252.76,110.75,0.00),v40,z0,tPen\WObj:=wPaper;
    MoveL Offs(pOrigin,251.91,110.40,0.00),v40,z0,tPen\WObj:=wPaper;
    MoveL Offs(pOrigin,250.43,110.40,0.00),v40,fine,tPen\WObj:=wPaper;
    MoveL Offs(pOrigin,250.43,110.40,6.00),v60,z5,tPen\WObj:=wPaper;
    MoveL Offs(pOrigin,252.21,109.44,6.00),vTravel,z5,tPen\WObj:=wPaper;
    MoveL Offs(pOrigin,252.21,109.44,0.00),v60,z0,tPen\WObj:=wPaper;
    MoveL Offs(pOrigin,247.55,114.10,0.00),v40,z0,tPen\WObj:=wPaper;
    MoveL Offs(pOrigin,248.00,115.15,0.00),v40,z0,tPen\WObj:=wPaper;
    MoveL Offs(pOrigin,253.11,110.04,0.00),v40,z0,tPen\WObj:=wPaper;
    MoveL Offs(pOrigin,254.00,110.64,0.00),v40,z0,tPen\WObj:=wPaper;
    MoveL Offs(pOrigin,248.75,115.90,0.00),v40,z0,tPen\WObj:=wPaper;
    MoveL Offs(pOrigin,249.64,116.49,0.00),v40,z0,tPen\WObj:=wPaper;
    MoveL Offs(pOrigin,254.60,111.53,0.00),v40,fine,tPen\WObj:=wPaper;
    MoveL Offs(pOrigin,254.60,111.53,6.00),v60,z5,tPen\WObj:=wPaper;
    MoveL Offs(pOrigin,254.90,112.73,6.00),vTravel,z5,tPen\WObj:=wPaper;
    MoveL Offs(pOrigin,254.90,112.73,0.00),v60,z0,tPen\WObj:=wPaper;
    MoveL Offs(pOrigin,250.69,116.94,0.00),v40,fine,tPen\WObj:=wPaper;
    MoveL Offs(pOrigin,250.69,116.94,6.00),v60,z5,tPen\WObj:=wPaper;
    MoveL Offs(pOrigin,252.34,116.78,6.00),vTravel,z5,tPen\WObj:=wPaper;
    MoveL Offs(pOrigin,252.34,116.78,0.00),v60,z0,tPen\WObj:=wPaper;
    MoveL Offs(pOrigin,254.59,114.53,0.00),v40,fine,tPen\WObj:=wPaper;
    MoveL Offs(pOrigin,254.59,114.53,6.00),v60,z5,tPen\WObj:=wPaper;
  ENDPROC

  PROC DrawPart252()
    MoveL Offs(pOrigin,253.19,115.07,6.00),vTravel,z5,tPen\WObj:=wPaper;
    MoveL Offs(pOrigin,253.19,115.07,0.00),v60,z0,tPen\WObj:=wPaper;
    MoveL Offs(pOrigin,252.76,115.50,0.00),v40,z0,tPen\WObj:=wPaper;
    MoveL Offs(pOrigin,253.19,115.07,0.00),v40,fine,tPen\WObj:=wPaper;
    MoveL Offs(pOrigin,253.19,115.07,6.00),v60,z5,tPen\WObj:=wPaper;
    MoveL Offs(pOrigin,250.43,113.80,6.00),vTravel,z5,tPen\WObj:=wPaper;
    MoveL Offs(pOrigin,250.43,113.80,0.00),v60,z0,tPen\WObj:=wPaper;
    MoveL Offs(pOrigin,251.70,113.59,0.00),v40,z0,tPen\WObj:=wPaper;
    MoveL Offs(pOrigin,251.49,112.81,0.00),v40,z0,tPen\WObj:=wPaper;
    MoveL Offs(pOrigin,250.64,112.74,0.00),v40,fine,tPen\WObj:=wPaper;
    MoveL Offs(pOrigin,250.64,112.74,6.00),v60,z5,tPen\WObj:=wPaper;
    MoveL Offs(pOrigin,231.51,91.03,6.00),vTravel,z5,tPen\WObj:=wPaper;
    MoveL Offs(pOrigin,231.51,91.03,0.00),v60,z0,tPen\WObj:=wPaper;
    MoveL Offs(pOrigin,230.24,91.03,0.00),v40,z0,tPen\WObj:=wPaper;
    MoveL Offs(pOrigin,230.24,89.98,0.00),v40,z0,tPen\WObj:=wPaper;
    MoveL Offs(pOrigin,231.30,89.98,0.00),v40,fine,tPen\WObj:=wPaper;
    MoveL Offs(pOrigin,231.30,89.98,6.00),v60,z5,tPen\WObj:=wPaper;
    MoveL Offs(pOrigin,232.35,88.98,6.00),vTravel,z5,tPen\WObj:=wPaper;
    MoveL Offs(pOrigin,232.35,88.98,0.00),v60,z0,tPen\WObj:=wPaper;
    MoveL Offs(pOrigin,229.35,91.99,0.00),v40,fine,tPen\WObj:=wPaper;
    MoveL Offs(pOrigin,229.35,91.99,6.00),v60,z5,tPen\WObj:=wPaper;
    MoveL Offs(pOrigin,229.05,89.29,6.00),vTravel,z5,tPen\WObj:=wPaper;
    MoveL Offs(pOrigin,229.05,89.29,0.00),v60,z0,tPen\WObj:=wPaper;
    MoveL Offs(pOrigin,231.91,86.44,0.00),v40,fine,tPen\WObj:=wPaper;
    MoveL Offs(pOrigin,231.91,86.44,6.00),v60,z5,tPen\WObj:=wPaper;
    MoveL Offs(pOrigin,230.88,85.75,6.00),vTravel,z5,tPen\WObj:=wPaper;
    MoveL Offs(pOrigin,230.88,85.75,0.00),v60,z0,tPen\WObj:=wPaper;
    MoveL Offs(pOrigin,229.60,85.75,0.00),v40,fine,tPen\WObj:=wPaper;
    MoveL Offs(pOrigin,229.60,85.75,6.00),v60,z5,tPen\WObj:=wPaper;
    MoveL Offs(pOrigin,228.61,86.75,6.00),vTravel,z5,tPen\WObj:=wPaper;
    MoveL Offs(pOrigin,228.61,86.75,0.00),v60,z0,tPen\WObj:=wPaper;
    MoveL Offs(pOrigin,231.92,83.44,0.00),v40,fine,tPen\WObj:=wPaper;
    MoveL Offs(pOrigin,231.92,83.44,6.00),v60,z5,tPen\WObj:=wPaper;
    MoveL Offs(pOrigin,230.88,82.14,6.00),vTravel,z5,tPen\WObj:=wPaper;
    MoveL Offs(pOrigin,230.88,82.14,0.00),v60,z0,tPen\WObj:=wPaper;
    MoveL Offs(pOrigin,230.24,81.29,0.00),v40,z0,tPen\WObj:=wPaper;
    MoveL Offs(pOrigin,227.69,67.05,0.00),v40,z0,tPen\WObj:=wPaper;
    MoveL Offs(pOrigin,227.69,66.74,0.00),v40,z0,tPen\WObj:=wPaper;
    MoveL Offs(pOrigin,225.99,66.74,0.00),v40,fine,tPen\WObj:=wPaper;
    MoveL Offs(pOrigin,225.99,66.74,6.00),v60,z5,tPen\WObj:=wPaper;
    MoveL Offs(pOrigin,226.41,68.86,6.00),vTravel,z5,tPen\WObj:=wPaper;
    MoveL Offs(pOrigin,226.41,68.86,0.00),v60,z0,tPen\WObj:=wPaper;
    MoveL Offs(pOrigin,227.90,68.86,0.00),v40,z0,tPen\WObj:=wPaper;
    MoveL Offs(pOrigin,228.11,69.91,0.00),v40,z0,tPen\WObj:=wPaper;
    MoveL Offs(pOrigin,226.84,69.91,0.00),v40,fine,tPen\WObj:=wPaper;
    MoveL Offs(pOrigin,226.84,69.91,6.00),v60,z5,tPen\WObj:=wPaper;
    MoveL Offs(pOrigin,225.37,69.08,6.00),vTravel,z5,tPen\WObj:=wPaper;
    MoveL Offs(pOrigin,225.37,69.08,0.00),v60,z0,tPen\WObj:=wPaper;
    MoveL Offs(pOrigin,229.43,65.02,0.00),v40,fine,tPen\WObj:=wPaper;
    MoveL Offs(pOrigin,229.43,65.02,6.00),v60,z5,tPen\WObj:=wPaper;
    MoveL Offs(pOrigin,229.89,60.08,6.00),vTravel,z5,tPen\WObj:=wPaper;
    MoveL Offs(pOrigin,229.89,60.08,0.00),v60,z0,tPen\WObj:=wPaper;
    MoveL Offs(pOrigin,235.30,54.67,0.00),v40,fine,tPen\WObj:=wPaper;
    MoveL Offs(pOrigin,235.30,54.67,6.00),v60,z5,tPen\WObj:=wPaper;
    MoveL Offs(pOrigin,225.26,55.75,6.00),vTravel,z5,tPen\WObj:=wPaper;
    MoveL Offs(pOrigin,225.26,55.75,0.00),v60,z0,tPen\WObj:=wPaper;
    MoveL Offs(pOrigin,222.71,58.30,0.00),v40,z0,tPen\WObj:=wPaper;
    MoveL Offs(pOrigin,223.65,58.30,0.00),v40,z0,tPen\WObj:=wPaper;
    MoveL Offs(pOrigin,224.92,58.30,0.00),v40,z0,tPen\WObj:=wPaper;
    MoveL Offs(pOrigin,224.71,57.24,0.00),v40,z0,tPen\WObj:=wPaper;
    MoveL Offs(pOrigin,223.44,57.24,0.00),v40,z0,tPen\WObj:=wPaper;
    MoveL Offs(pOrigin,223.01,56.18,0.00),v40,z0,tPen\WObj:=wPaper;
    MoveL Offs(pOrigin,224.50,56.18,0.00),v40,z0,tPen\WObj:=wPaper;
    MoveL Offs(pOrigin,224.08,55.13,0.00),v40,z0,tPen\WObj:=wPaper;
    MoveL Offs(pOrigin,222.80,55.13,0.00),v40,z0,tPen\WObj:=wPaper;
    MoveL Offs(pOrigin,222.38,54.07,0.00),v40,z0,tPen\WObj:=wPaper;
    MoveL Offs(pOrigin,223.65,54.07,0.00),v40,z0,tPen\WObj:=wPaper;
    MoveL Offs(pOrigin,224.52,53.50,0.00),v40,z0,tPen\WObj:=wPaper;
    MoveL Offs(pOrigin,221.82,56.21,0.00),v40,fine,tPen\WObj:=wPaper;
    MoveL Offs(pOrigin,221.82,56.21,6.00),v60,z5,tPen\WObj:=wPaper;
    MoveL Offs(pOrigin,221.95,53.02,6.00),vTravel,z5,tPen\WObj:=wPaper;
    MoveL Offs(pOrigin,221.95,53.02,0.00),v60,z0,tPen\WObj:=wPaper;
    MoveL Offs(pOrigin,223.44,53.02,0.00),v40,fine,tPen\WObj:=wPaper;
    MoveL Offs(pOrigin,223.44,53.02,6.00),v60,z5,tPen\WObj:=wPaper;
    MoveL Offs(pOrigin,223.16,48.72,6.00),vTravel,z5,tPen\WObj:=wPaper;
    MoveL Offs(pOrigin,223.16,48.72,0.00),v60,z0,tPen\WObj:=wPaper;
    MoveL Offs(pOrigin,215.05,40.61,0.00),v40,z0,tPen\WObj:=wPaper;
    MoveL Offs(pOrigin,214.08,40.05,0.00),v40,z0,tPen\WObj:=wPaper;
    MoveL Offs(pOrigin,210.02,44.11,0.00),v40,fine,tPen\WObj:=wPaper;
    MoveL Offs(pOrigin,210.02,44.11,6.00),v60,z5,tPen\WObj:=wPaper;
    MoveL Offs(pOrigin,210.16,42.82,6.00),vTravel,z5,tPen\WObj:=wPaper;
    MoveL Offs(pOrigin,210.16,42.82,0.00),v60,z0,tPen\WObj:=wPaper;
    MoveL Offs(pOrigin,210.16,41.34,0.00),v40,fine,tPen\WObj:=wPaper;
    MoveL Offs(pOrigin,210.16,41.34,6.00),v60,z5,tPen\WObj:=wPaper;
    MoveL Offs(pOrigin,210.93,40.21,6.00),vTravel,z5,tPen\WObj:=wPaper;
    MoveL Offs(pOrigin,210.93,40.21,0.00),v60,z0,tPen\WObj:=wPaper;
    MoveL Offs(pOrigin,206.12,45.02,0.00),v40,z0,tPen\WObj:=wPaper;
    MoveL Offs(pOrigin,205.62,44.63,0.00),v40,z0,tPen\WObj:=wPaper;
    MoveL Offs(pOrigin,204.12,43.12,0.00),v40,z0,tPen\WObj:=wPaper;
    MoveL Offs(pOrigin,203.25,43.51,0.00),v40,z0,tPen\WObj:=wPaper;
    MoveL Offs(pOrigin,207.29,43.51,0.00),v40,z0,tPen\WObj:=wPaper;
    MoveL Offs(pOrigin,208.02,44.03,0.00),v40,z0,tPen\WObj:=wPaper;
    MoveL Offs(pOrigin,206.36,42.38,0.00),v40,z0,tPen\WObj:=wPaper;
    MoveL Offs(pOrigin,205.32,42.83,0.00),v40,z0,tPen\WObj:=wPaper;
    MoveL Offs(pOrigin,206.67,44.18,0.00),v40,fine,tPen\WObj:=wPaper;
    MoveL Offs(pOrigin,206.67,44.18,6.00),v60,z5,tPen\WObj:=wPaper;
    MoveL Offs(pOrigin,208.07,44.57,6.00),vTravel,z5,tPen\WObj:=wPaper;
    MoveL Offs(pOrigin,208.07,44.57,0.00),v60,z0,tPen\WObj:=wPaper;
    MoveL Offs(pOrigin,212.58,40.06,0.00),v40,fine,tPen\WObj:=wPaper;
    MoveL Offs(pOrigin,212.58,40.06,6.00),v60,z5,tPen\WObj:=wPaper;
    MoveL Offs(pOrigin,208.14,41.40,6.00),vTravel,z5,tPen\WObj:=wPaper;
    MoveL Offs(pOrigin,208.14,41.40,0.00),v60,z0,tPen\WObj:=wPaper;
    MoveL Offs(pOrigin,227.90,41.40,0.00),v40,z0,tPen\WObj:=wPaper;
    MoveL Offs(pOrigin,228.23,41.85,0.00),v40,z0,tPen\WObj:=wPaper;
    MoveL Offs(pOrigin,226.13,39.75,0.00),v40,z0,tPen\WObj:=wPaper;
    MoveL Offs(pOrigin,226.00,40.49,0.00),v40,z0,tPen\WObj:=wPaper;
    MoveL Offs(pOrigin,226.00,43.04,0.00),v40,z0,tPen\WObj:=wPaper;
    MoveL Offs(pOrigin,226.20,43.51,0.00),v40,z0,tPen\WObj:=wPaper;
    MoveL Offs(pOrigin,221.74,43.51,0.00),v40,z0,tPen\WObj:=wPaper;
    MoveL Offs(pOrigin,221.95,43.46,0.00),v40,z0,tPen\WObj:=wPaper;
    MoveL Offs(pOrigin,222.59,42.97,0.00),v40,z0,tPen\WObj:=wPaper;
    MoveL Offs(pOrigin,224.50,42.40,0.00),v40,z0,tPen\WObj:=wPaper;
    MoveL Offs(pOrigin,224.71,43.04,0.00),v40,z0,tPen\WObj:=wPaper;
    MoveL Offs(pOrigin,224.93,43.25,0.00),v40,z0,tPen\WObj:=wPaper;
    MoveL Offs(pOrigin,224.50,43.67,0.00),v40,z0,tPen\WObj:=wPaper;
    MoveL Offs(pOrigin,224.71,43.04,0.00),v40,z0,tPen\WObj:=wPaper;
    MoveL Offs(pOrigin,224.93,43.25,0.00),v40,z0,tPen\WObj:=wPaper;
    MoveL Offs(pOrigin,224.50,43.67,0.00),v40,z0,tPen\WObj:=wPaper;
    MoveL Offs(pOrigin,224.71,43.04,0.00),v40,fine,tPen\WObj:=wPaper;
    MoveL Offs(pOrigin,224.71,43.04,6.00),v60,z5,tPen\WObj:=wPaper;
  ENDPROC

